	(*Reposition Request#3*)
	(*Pick Up repo*)
	IF (MAIN.R4.Peripheral_Req.2 AND (MAIN.R4.Task_ID_Ack=Pickup_Fix102))
		THEN
			Repo_Reqs.2:= TRUE;
	END_IF;

	(*Reposition Request#4*)
	IF FALSE
		THEN
			Repo_Reqs.3:= TRUE;
	END_IF;

	(*Reposition Request#5*)
	IF FALSE
		THEN
			Repo_Reqs.4:= TRUE;
	END_IF;

	(*Reposition Request#6*)
	IF FALSE
		THEN
			Repo_Reqs.5:= TRUE;
	END_IF;

	(*Reposition Request#7*)
	IF FALSE
		THEN
			Repo_Reqs.6:= TRUE;
	END_IF;

	(*Reposition Request#8*)
	IF FALSE
		THEN
			Repo_Reqs.7:= TRUE;
	END_IF;

	(*Reset All Reposition Acks At the End Of Cycle*)
	IF Cycle_Complete
		THEN
			Repo_Reqs:= 0;
	END_IF;

(*------------------------- Reposition Acks ---------------------*)
	Repo_Ack.0:= Repo_Reqs.0 AND Tool_At_Load.0;   (*Drop Off*)
	Repo_Ack.1:= Repo_Reqs.1 AND FALSE;            (*Inspection*)
	Repo_Ack.2:= Repo_Reqs.2 AND Tool_At_Unload.1; (*Pick Up*)
	Repo_Ack.3:= Repo_Reqs.3 AND FALSE;
	Repo_Ack.4:= Repo_Reqs.4 AND FALSE;
	Repo_Ack.5:= Repo_Reqs.5 AND FALSE;
	Repo_Ack.6:= Repo_Reqs.6 AND FALSE;
	Repo_Ack.7:= Repo_Reqs.7 AND FALSE;
END_ACTION

ACTION ValveBank1:


(*+++++++++++THIS AREA IS CUSTOM PER INSTALLATION AND WILL HAVE TO BE MODIFIED PER +++++++++++++*)
(*+++++++++++THIS AREA IS CUSTOM PER INSTALLATION AND WILL HAVE TO BE MODIFIED PER +++++++++++++*)
(*+++++++++++THIS AREA IS CUSTOM PER INSTALLATION AND WILL HAVE TO BE MODIFIED PER +++++++++++++*)

(*+++++++++++VALVE BANK 1 +++++++++++++*)
(*+++++++++++VALVE BANK 1 +++++++++++++*)
(*+++++++++++VALVE BANK 1 +++++++++++++*)


	(*Valve 1, A+B*)
	// NOW Pin 1,2 Piped and Labled From Supplier (*TLK*)
		Valve1FB
			(
			Enable_Motion:= Enable_Motion ,
			Enable_Latch:= TRUE,					(*Enabling Runs Valve as detent type (maintained solenoids*)
			Enable_SideA_PreCharge:= FALSE,		(*Enabling Turns Side A PreCharge Active, reset when Side B is energized in Auto*)
			Enable_SideB_PreCharge:= FALSE,		(*Enabling Turns Side B PreCharge Active, reset when Side A is energized in Auto*)
			PreCharge_Time:= T#0.1S,
			Enable_Auto_Commands:= In_Auto,
			Enable_Manual_Commands:= In_Manual AND All_Robots_Clear,
			In_Manual_SideA_Command:= Discrete_In.ManReqs.0,
			In_Manual_SideB_Command:= (Discrete_In.ManReqs.1 OR Discrete_In.Go_Home),
			SideA_Indicator:= (Pin1ADVD AND Pin2ADVD) OR Manual_Ind_HomePrompt,
			SideB_Indicator:= (Pin1RETD AND Pin2RETD),
			TurnOn_SideA_SOL=> N100.Q.0,
			TurnOn_SideB_SOL=> N100.Q.1,
			TurnOn_SideA_Indicator=> Manual_Indicators1.0,
			TurnOn_SideB_Indicator=> Manual_Indicators1.1
			 );
		Valve1FB.In_Auto_SideA_Command:= (*Clamp_Step.1 AND NOT Unclamp_Step.1;*) Clamp_Step.0 AND NOT Unclamp_Step.0;
		Valve1FB.In_Auto_SideB_Command:= (*NOT Clamp_Step.1 AND Unclamp_Step.1;*) NOT Clamp_Step.0 AND Unclamp_Step.0;


	(*Valve 2, A+B*)
	// NOW Clamp 1,2,3,4 Piped and Labled From Supplier (*TLK*)
		Valve2FB
			(
			Enable_Motion:= Enable_Motion ,
			Enable_Latch:= TRUE,					(*Enabling Runs Valve as detent type (maintained solenoids*)
			Enable_SideA_PreCharge:= FALSE,		(*Enabling Turns Side A PreCharge Active, reset when Side B is energized in Auto*)
			Enable_SideB_PreCharge:= FALSE,		(*Enabling Turns Side B PreCharge Active, reset when Side A is energized in Auto*)
			PreCharge_Time:= T#0.10S,
			Enable_Auto_Commands:= In_Auto,
			Enable_Manual_Commands:= In_Manual AND All_Robots_Clear,
			In_Manual_SideA_Command:= (Discrete_In.ManReqs.2 OR Discrete_In.Go_Home),
			In_Manual_SideB_Command:= Discrete_In.ManReqs.3,		
			SideA_Indicator:= (Clamp1ADVD AND Clamp2ADVD AND Clamp3ADVD AND Clamp4ADVD),
			SideB_Indicator:= (Clamp1RETD AND Clamp2RETD AND Clamp3RETD AND Clamp4RETD) OR Manual_Ind_HomePrompt,
			TurnOn_SideA_SOL=> N100.Q.2,
			TurnOn_SideB_SOL=> N100.Q.3,
			TurnOn_SideA_Indicator=> Manual_Indicators1.2,
			TurnOn_SideB_Indicator=> Manual_Indicators1.3
			 );
		Valve2FB.In_Auto_SideA_Command:= (*Clamp_Step.0 AND NOT Unclamp_Step.0;*) Clamp_Step.1 AND NOT Unclamp_Step.1;
		Valve2FB.In_Auto_SideB_Command:= (*NOT Clamp_Step.0 AND Unclamp_Step.0;*) NOT Clamp_Step.1 AND Unclamp_Step.1;


		
		
		
		
		
		
		
		
		
		
		
		
		
		
		
		
		
		
		
	(*Valve 3, A+B*)
	(*spare*)
		Valve3FB
			(
			Enable_Motion:= Enable_Motion ,
			Enable_Latch:= TRUE,					(*Enabling Runs Valve as detent type (maintained solenoids*)
			Enable_SideA_PreCharge:= FALSE,		(*Enabling Turns Side A PreCharge Active, reset when Side B is energized in Auto*)
			Enable_SideB_PreCharge:= FALSE,		(*Enabling Turns Side B PreCharge Active, reset when Side A is energized in Auto*)
			PreCharge_Time:= T#0.10S,
			Enable_Auto_Commands:= In_Auto,
			Enable_Manual_Commands:= In_Manual AND All_Robots_Clear,
			In_Manual_SideA_Command:= Discrete_In.ManReqs.4,
			In_Manual_SideB_Command:= Discrete_In.ManReqs.5,
			SideA_Indicator:= FALSE,
			SideB_Indicator:= FALSE,
			TurnOn_SideA_SOL=> N100.Q.4,
			TurnOn_SideB_SOL=> N100.Q.5,
			TurnOn_SideA_Indicator=> Manual_Indicators1.4,
			TurnOn_SideB_Indicator=> Manual_Indicators1.5
			 );
		Valve3FB.In_Auto_SideA_Command:= FALSE;
		Valve3FB.In_Auto_SideB_Command:= FALSE;



(*end*)
END_ACTION

ACTION ValveBank2:


(*+++++++++++THIS AREA IS CUSTOM PER INSTALLATION AND WILL HAVE TO BE MODIFIED PER +++++++++++++*)
(*+++++++++++THIS AREA IS CUSTOM PER INSTALLATION AND WILL HAVE TO BE MODIFIED PER +++++++++++++*)
(*+++++++++++THIS AREA IS CUSTOM PER INSTALLATION AND WILL HAVE TO BE MODIFIED PER +++++++++++++*)

(*+++++++++++VALVE BANK 2 +++++++++++++*)
(*+++++++++++VALVE BANK 2 +++++++++++++*)
(*+++++++++++VALVE BANK 2 +++++++++++++*)


	(*Valve 17, A+B*)
	(*spare*)
		Valve17FB
			(
			Enable_Motion:= Enable_Motion ,
			Enable_Latch:= TRUE,					(*Enabling Runs Valve as detent type (maintained solenoids*)
			Enable_SideA_PreCharge:= FALSE,		(*Enabling Turns Side A PreCharge Active, reset when Side B is energized in Auto*)
			Enable_SideB_PreCharge:= FALSE,		(*Enabling Turns Side B PreCharge Active, reset when Side A is energized in Auto*)
			PreCharge_Time:= T#0.1S,
			Enable_Auto_Commands:= In_Auto,
			Enable_Manual_Commands:= In_Manual AND All_Robots_Clear,
			In_Manual_SideA_Command:= Discrete_In.ManReqs2.0,
			In_Manual_SideB_Command:= (Discrete_In.ManReqs2.1 OR Discrete_In.Go_Home),
			SideA_Indicator:= FALSE,
			SideB_Indicator:= FALSE,
			TurnOn_SideA_SOL=> N101.Q.0,
			TurnOn_SideB_SOL=> N101.Q.1,
			TurnOn_SideA_Indicator=> Manual_Indicators2.0,
			TurnOn_SideB_Indicator=> Manual_Indicators2.1
			 );
		Valve17FB.In_Auto_SideA_Command:= FALSE;
		Valve17FB.In_Auto_SideB_Command:= FALSE;


	(*Valve 18, A+B*)
	(*spare*)
		Valve18FB
			(
			Enable_Motion:= Enable_Motion ,
			Enable_Latch:= TRUE,					(*Enabling Runs Valve as detent type (maintained solenoids*)
			Enable_SideA_PreCharge:= FALSE,		(*Enabling Turns Side A PreCharge Active, reset when Side B is energized in Auto*)
			Enable_SideB_PreCharge:= FALSE,		(*Enabling Turns Side B PreCharge Active, reset when Side A is energized in Auto*)
			PreCharge_Time:= T#0.10S,
			Enable_Auto_Commands:= In_Auto,
			Enable_Manual_Commands:= In_Manual AND All_Robots_Clear,
			In_Manual_SideA_Command:= Discrete_In.ManReqs2.2,
			In_Manual_SideB_Command:= Discrete_In.ManReqs2.3,
			SideA_Indicator:= FALSE,
			SideB_Indicator:= FALSE,
			TurnOn_SideA_SOL=> N101.Q.2,
			TurnOn_SideB_SOL=> N101.Q.3,
			TurnOn_SideA_Indicator=> Manual_Indicators2.2,
			TurnOn_SideB_Indicator=> Manual_Indicators2.3
			 );
		Valve18FB.In_Auto_SideA_Command:= FALSE;
		Valve18FB.In_Auto_SideB_Command:= FALSE;

	(*Valve 19, A+B*)
	(*spare*)
		Valve19FB
			(
			Enable_Motion:= Enable_Motion ,
			Enable_Latch:= TRUE,					(*Enabling Runs Valve as detent type (maintained solenoids*)
			Enable_SideA_PreCharge:= FALSE,		(*Enabling Turns Side A PreCharge Active, reset when Side B is energized in Auto*)
			Enable_SideB_PreCharge:= FALSE,		(*Enabling Turns Side B PreCharge Active, reset when Side A is energized in Auto*)
			PreCharge_Time:= T#0.10S,
			Enable_Auto_Commands:= In_Auto,
			Enable_Manual_Commands:= In_Manual AND All_Robots_Clear,
			In_Manual_SideA_Command:= Discrete_In.ManReqs2.4,
			In_Manual_SideB_Command:= Discrete_In.ManReqs2.5,
			SideA_Indicator:= FALSE,
			SideB_Indicator:= FALSE,
			TurnOn_SideA_SOL=> N101.Q.4,
			TurnOn_SideB_SOL=> N101.Q.5,
			TurnOn_SideA_Indicator=> Manual_Indicators2.4,
			TurnOn_SideB_Indicator=> Manual_Indicators2.5
			 );
		Valve19FB.In_Auto_SideA_Command:= FALSE;
		Valve19FB.In_Auto_SideB_Command:= FALSE;


	(*Valve 20, A+B*)
	(*spare*)
		Valve20FB
			(
			Enable_Motion:= Enable_Motion ,
			Enable_Latch:= TRUE,					(*Enabling Runs Valve as detent type (maintained solenoids*)
			Enable_SideA_PreCharge:= FALSE,		(*Enabling Turns Side A PreCharge Active, reset when Side B is energized in Auto*)
			Enable_SideB_PreCharge:= FALSE,		(*Enabling Turns Side B PreCharge Active, reset when Side A is energized in Auto*)
			PreCharge_Time:= T#0.10S,
			Enable_Auto_Commands:= In_Auto,
			Enable_Manual_Commands:= In_Manual AND All_Robots_Clear,
			In_Manual_SideA_Command:= Discrete_In.ManReqs2.6,
			In_Manual_SideB_Command:= Discrete_In.ManReqs2.7,
			SideA_Indicator:= FALSE,
			SideB_Indicator:= FALSE,
			TurnOn_SideA_SOL=> N101.Q.6,
			TurnOn_SideB_SOL=> N101.Q.7,
			TurnOn_SideA_Indicator=> Manual_Indicators2.6,
			TurnOn_SideB_Indicator=> Manual_Indicators2.7
			 );
		Valve20FB.In_Auto_SideA_Command:= FALSE;
		Valve20FB.In_Auto_SideB_Command:= FALSE;


	(*Valve 21, A+B*)
	(*spare*)
		Valve21FB
			(
			Enable_Motion:= Enable_Motion ,
			Enable_Latch:= TRUE,					(*Enabling Runs Valve as detent type (maintained solenoids*)
			Enable_SideA_PreCharge:= FALSE,		(*Enabling Turns Side A PreCharge Active, reset when Side B is energized in Auto*)
			Enable_SideB_PreCharge:= FALSE,		(*Enabling Turns Side B PreCharge Active, reset when Side A is energized in Auto*)
			PreCharge_Time:= T#0.10S,
			Enable_Auto_Commands:= In_Auto,
			Enable_Manual_Commands:= In_Manual AND All_Robots_Clear,
			In_Manual_SideA_Command:= Discrete_In.ManReqs2.8,
			In_Manual_SideB_Command:= Discrete_In.ManReqs2.9,
			SideA_Indicator:= FALSE,
			SideB_Indicator:= FALSE,
			TurnOn_SideA_SOL=> N101.Q.8,
			TurnOn_SideB_SOL=> N101.Q.9,
			TurnOn_SideA_Indicator=> Manual_Indicators2.8,
			TurnOn_SideB_Indicator=> Manual_Indicators2.9
			 );
		Valve21FB.In_Auto_SideA_Command:= FALSE;
		Valve21FB.In_Auto_SideB_Command:= FALSE;


	(*Valve 22, A+B*)
	(*spare*)
		Valve22FB
			(
			Enable_Motion:= Enable_Motion ,
			Enable_Latch:= TRUE,					(*Enabling Runs Valve as detent type (maintained solenoids*)
			Enable_SideA_PreCharge:= FALSE,		(*Enabling Turns Side A PreCharge Active, reset when Side B is energized in Auto*)
			Enable_SideB_PreCharge:= FALSE,		(*Enabling Turns Side B PreCharge Active, reset when Side A is energized in Auto*)
			PreCharge_Time:= T#0.10S,
			Enable_Auto_Commands:= In_Auto,
			Enable_Manual_Commands:= In_Manual AND All_Robots_Clear,
			In_Manual_SideA_Command:= Discrete_In.ManReqs2.10,
			In_Manual_SideB_Command:= Discrete_In.ManReqs2.11,
			SideA_Indicator:= FALSE,
			SideB_Indicator:= FALSE,
			TurnOn_SideA_SOL=> N101.Q.10,
			TurnOn_SideB_SOL=> N101.Q.11,
			TurnOn_SideA_Indicator=> Manual_Indicators2.10,
			TurnOn_SideB_Indicator=> Manual_Indicators2.11
			 );
		Valve22FB.In_Auto_SideA_Command:= FALSE;
		Valve22FB.In_Auto_SideB_Command:= FALSE;


	(*Valve 23, A+B*)
	(*spare*)
		Valve23FB
			(
			Enable_Motion:= Enable_Motion ,
			Enable_Latch:= TRUE,					(*Enabling Runs Valve as detent type (maintained solenoids*)
			Enable_SideA_PreCharge:= FALSE,		(*Enabling Turns Side A PreCharge Active, reset when Side B is energized in Auto*)
			Enable_SideB_PreCharge:= FALSE,		(*Enabling Turns Side B PreCharge Active, reset when Side A is energized in Auto*)
			PreCharge_Time:= T#0.10S,
			Enable_Auto_Commands:= In_Auto,
			Enable_Manual_Commands:= In_Manual AND All_Robots_Clear,
			In_Manual_SideA_Command:= Discrete_In.ManReqs2.12,
			In_Manual_SideB_Command:= Discrete_In.ManReqs2.13,
			SideA_Indicator:= FALSE,
			SideB_Indicator:= FALSE,
			TurnOn_SideA_SOL=> N101.Q.12,
			TurnOn_SideB_SOL=> N101.Q.13,
			TurnOn_SideA_Indicator=> Manual_Indicators2.12,
			TurnOn_SideB_Indicator=> Manual_Indicators2.13
			 );
		Valve23FB.In_Auto_SideA_Command:= FALSE;
		Valve23FB.In_Auto_SideB_Command:= FALSE;


	(*Valve 24, A+B*)
	(*spare*)
		Valve24FB
			(
			Enable_Motion:= Enable_Motion ,
			Enable_Latch:= TRUE,					(*Enabling Runs Valve as detent type (maintained solenoids*)
			Enable_SideA_PreCharge:= FALSE,		(*Enabling Turns Side A PreCharge Active, reset when Side B is energized in Auto*)
			Enable_SideB_PreCharge:= FALSE,		(*Enabling Turns Side B PreCharge Active, reset when Side A is energized in Auto*)
			PreCharge_Time:= T#0.10S,
			Enable_Auto_Commands:= In_Auto,
			Enable_Manual_Commands:= In_Manual AND All_Robots_Clear,
			In_Manual_SideA_Command:= Discrete_In.ManReqs2.14,
			In_Manual_SideB_Command:= Discrete_In.ManReqs2.15,
			SideA_Indicator:= FALSE,
			SideB_Indicator:= FALSE,
			TurnOn_SideA_SOL=> N101.Q.14,
			TurnOn_SideB_SOL=> N101.Q.15,
			TurnOn_SideA_Indicator=> Manual_Indicators2.14,
			TurnOn_SideB_Indicator=> Manual_Indicators2.15
			 );
		Valve24FB.In_Auto_SideA_Command:= FALSE;
		Valve24FB.In_Auto_SideB_Command:= FALSE;


	(*Valve 25, A+B*)
	(*spare*)
		Valve25FB
			(
			Enable_Motion:= Enable_Motion ,
			Enable_Latch:= TRUE,					(*Enabling Runs Valve as detent type (maintained solenoids*)
			Enable_SideA_PreCharge:= FALSE,		(*Enabling Turns Side A PreCharge Active, reset when Side B is energized in Auto*)
			Enable_SideB_PreCharge:= FALSE,		(*Enabling Turns Side B PreCharge Active, reset when Side A is energized in Auto*)
			PreCharge_Time:= T#0.10S,
			Enable_Auto_Commands:= In_Auto,
			Enable_Manual_Commands:= In_Manual AND All_Robots_Clear,
			In_Manual_SideA_Command:= Discrete_In.ManReqs2.16,
			In_Manual_SideB_Command:= Discrete_In.ManReqs2.17,
			SideA_Indicator:= FALSE,
			SideB_Indicator:= FALSE,
			TurnOn_SideA_SOL=> N101.Q.16,
			TurnOn_SideB_SOL=> N101.Q.17,
			TurnOn_SideA_Indicator=> Manual_Indicators2.16,
			TurnOn_SideB_Indicator=> Manual_Indicators2.17
			 );
		Valve25FB.In_Auto_SideA_Command:= FALSE;
		Valve25FB.In_Auto_SideB_Command:= FALSE;


	(*Valve 26, A+B*)
	(*spare*)
		Valve26FB
			(
			Enable_Motion:= Enable_Motion ,
			Enable_Latch:= TRUE,					(*Enabling Runs Valve as detent type (maintained solenoids*)
			Enable_SideA_PreCharge:= FALSE,		(*Enabling Turns Side A PreCharge Active, reset when Side B is energized in Auto*)
			Enable_SideB_PreCharge:= FALSE,		(*Enabling Turns Side B PreCharge Active, reset when Side A is energized in Auto*)
			PreCharge_Time:= T#0.10S,
			Enable_Auto_Commands:= In_Auto,
			Enable_Manual_Commands:= In_Manual AND All_Robots_Clear,
			In_Manual_SideA_Command:= Discrete_In.ManReqs2.18,
			In_Manual_SideB_Command:= Discrete_In.ManReqs2.19,
			SideA_Indicator:= FALSE,
			SideB_Indicator:= FALSE,
			TurnOn_SideA_SOL=> N101.Q.18,
			TurnOn_SideB_SOL=> N101.Q.19,
			TurnOn_SideA_Indicator=> Manual_Indicators2.18,
			TurnOn_SideB_Indicator=> Manual_Indicators2.19
			 );
		Valve26FB.In_Auto_SideA_Command:= FALSE;
		Valve26FB.In_Auto_SideB_Command:= FALSE;


	(*Valve 27, A+B*)
	(*spare*)
		Valve27FB
			(
			Enable_Motion:= Enable_Motion ,
			Enable_Latch:= TRUE,					(*Enabling Runs Valve as detent type (maintained solenoids*)
			Enable_SideA_PreCharge:= FALSE,		(*Enabling Turns Side A PreCharge Active, reset when Side B is energized in Auto*)
			Enable_SideB_PreCharge:= FALSE,		(*Enabling Turns Side B PreCharge Active, reset when Side A is energized in Auto*)
			PreCharge_Time:= T#0.10S,
			Enable_Auto_Commands:= In_Auto,
			Enable_Manual_Commands:= In_Manual AND All_Robots_Clear,
			In_Manual_SideA_Command:= Discrete_In.ManReqs2.20,
			In_Manual_SideB_Command:= Discrete_In.ManReqs2.21,
			SideA_Indicator:= FALSE,
			SideB_Indicator:= FALSE,
			TurnOn_SideA_SOL=> N101.Q.20,
			TurnOn_SideB_SOL=> N101.Q.21,
			TurnOn_SideA_Indicator=> Manual_Indicators2.20,
			TurnOn_SideB_Indicator=> Manual_Indicators2.21
			 );
		Valve27FB.In_Auto_SideA_Command:= FALSE;
		Valve27FB.In_Auto_SideB_Command:= FALSE;


	(*Valve 28, A+B*)
	(*spare*)
		Valve28FB
			(
			Enable_Motion:= Enable_Motion ,
			Enable_Latch:= TRUE,					(*Enabling Runs Valve as detent type (maintained solenoids*)
			Enable_SideA_PreCharge:= FALSE,		(*Enabling Turns Side A PreCharge Active, reset when Side B is energized in Auto*)
			Enable_SideB_PreCharge:= FALSE,		(*Enabling Turns Side B PreCharge Active, reset when Side A is energized in Auto*)
			PreCharge_Time:= T#0.10S,
			Enable_Auto_Commands:= In_Auto,
			Enable_Manual_Commands:= In_Manual AND All_Robots_Clear,
			In_Manual_SideA_Command:= Discrete_In.ManReqs2.22,
			In_Manual_SideB_Command:= Discrete_In.ManReqs2.23,
			SideA_Indicator:= FALSE,
			SideB_Indicator:= FALSE,
			TurnOn_SideA_SOL=> N101.Q.22,
			TurnOn_SideB_SOL=> N101.Q.23,
			TurnOn_SideA_Indicator=> Manual_Indicators2.22,
			TurnOn_SideB_Indicator=> Manual_Indicators2.23
			 );
		Valve28FB.In_Auto_SideA_Command:= FALSE;
		Valve28FB.In_Auto_SideB_Command:= FALSE;


	(*Valve 29, A+B*)
	(*spare*)
		Valve29FB
			(
			Enable_Motion:= Enable_Motion ,
			Enable_Latch:= TRUE,					(*Enabling Runs Valve as detent type (maintained solenoids*)
			Enable_SideA_PreCharge:= FALSE,		(*Enabling Turns Side A PreCharge Active, reset when Side B is energized in Auto*)
			Enable_SideB_PreCharge:= FALSE,		(*Enabling Turns Side B PreCharge Active, reset when Side A is energized in Auto*)
			PreCharge_Time:= T#0.10S,
			Enable_Auto_Commands:= In_Auto,
			Enable_Manual_Commands:= In_Manual AND All_Robots_Clear,
			In_Manual_SideA_Command:= Discrete_In.ManReqs2.24,
			In_Manual_SideB_Command:= Discrete_In.ManReqs2.25,
			SideA_Indicator:= FALSE,
			SideB_Indicator:= FALSE,
			TurnOn_SideA_SOL=> N101.Q.24,
			TurnOn_SideB_SOL=> N101.Q.25,
			TurnOn_SideA_Indicator=> Manual_Indicators2.24,
			TurnOn_SideB_Indicator=> Manual_Indicators2.25
			 );
		Valve29FB.In_Auto_SideA_Command:= FALSE;
		Valve29FB.In_Auto_SideB_Command:= FALSE;


	(*Valve 30, A+B*)
	(*spare*)
		Valve30FB
			(
			Enable_Motion:= Enable_Motion ,
			Enable_Latch:= TRUE,					(*Enabling Runs Valve as detent type (maintained solenoids*)
			Enable_SideA_PreCharge:= FALSE,		(*Enabling Turns Side A PreCharge Active, reset when Side B is energized in Auto*)
			Enable_SideB_PreCharge:= FALSE,		(*Enabling Turns Side B PreCharge Active, reset when Side A is energized in Auto*)
			PreCharge_Time:= T#0.10S,
			Enable_Auto_Commands:= In_Auto,
			Enable_Manual_Commands:= In_Manual AND All_Robots_Clear,
			In_Manual_SideA_Command:= Discrete_In.ManReqs2.26,
			In_Manual_SideB_Command:= Discrete_In.ManReqs2.27,
			SideA_Indicator:= FALSE,
			SideB_Indicator:= FALSE,
			TurnOn_SideA_SOL=> N101.Q.26,
			TurnOn_SideB_SOL=> N101.Q.27,
			TurnOn_SideA_Indicator=> Manual_Indicators2.26,
			TurnOn_SideB_Indicator=> Manual_Indicators2.27
			 );
		Valve30FB.In_Auto_SideA_Command:= FALSE;
		Valve30FB.In_Auto_SideB_Command:= FALSE;


	(*Valve 31, A+B*)
	(*spare*)
		Valve31FB
			(
			Enable_Motion:= Enable_Motion ,
			Enable_Latch:= TRUE,					(*Enabling Runs Valve as detent type (maintained solenoids*)
			Enable_SideA_PreCharge:= FALSE,		(*Enabling Turns Side A PreCharge Active, reset when Side B is energized in Auto*)
			Enable_SideB_PreCharge:= FALSE,		(*Enabling Turns Side B PreCharge Active, reset when Side A is energized in Auto*)
			PreCharge_Time:= T#0.10S,
			Enable_Auto_Commands:= In_Auto,
			Enable_Manual_Commands:= In_Manual AND All_Robots_Clear,
			In_Manual_SideA_Command:= Discrete_In.ManReqs2.28,
			In_Manual_SideB_Command:= Discrete_In.ManReqs2.29,
			SideA_Indicator:= FALSE,
			SideB_Indicator:= FALSE,
			TurnOn_SideA_SOL=> N101.Q.28,
			TurnOn_SideB_SOL=> N101.Q.29,
			TurnOn_SideA_Indicator=> Manual_Indicators2.28,
			TurnOn_SideB_Indicator=> Manual_Indicators2.29
			 );
		Valve31FB.In_Auto_SideA_Command:= FALSE;
		Valve31FB.In_Auto_SideB_Command:= FALSE;


	(*Valve 32, A+B*)
	(*spare*)
		Valve32FB
			(
			Enable_Motion:= Enable_Motion ,
			Enable_Latch:= TRUE,					(*Enabling Runs Valve as detent type (maintained solenoids*)
			Enable_SideA_PreCharge:= FALSE,		(*Enabling Turns Side A PreCharge Active, reset when Side B is energized in Auto*)
			Enable_SideB_PreCharge:= FALSE,		(*Enabling Turns Side B PreCharge Active, reset when Side A is energized in Auto*)
			PreCharge_Time:= T#0.10S,
			Enable_Auto_Commands:= In_Auto,
			Enable_Manual_Commands:= In_Manual AND All_Robots_Clear,
			In_Manual_SideA_Command:= Discrete_In.ManReqs2.30,
			In_Manual_SideB_Command:= Discrete_In.ManReqs2.31,
			SideA_Indicator:= FALSE,
			SideB_Indicator:= FALSE,
			TurnOn_SideA_SOL=> N101.Q.30,
			TurnOn_SideB_SOL=> N101.Q.31,
			TurnOn_SideA_Indicator=> Manual_Indicators2.30,
			TurnOn_SideB_Indicator=> Manual_Indicators2.31
			 );
		Valve32FB.In_Auto_SideA_Command:= FALSE;
		Valve32FB.In_Auto_SideB_Command:= FALSE;




















(*end*)
END_ACTION

ACTION ValveBank3:


(*+++++++++++THIS AREA IS CUSTOM PER INSTALLATION AND WILL HAVE TO BE MODIFIED PER +++++++++++++*)
(*+++++++++++THIS AREA IS CUSTOM PER INSTALLATION AND WILL HAVE TO BE MODIFIED PER +++++++++++++*)
(*+++++++++++THIS AREA IS CUSTOM PER INSTALLATION AND WILL HAVE TO BE MODIFIED PER +++++++++++++*)

(*+++++++++++VALVE BANK 3 +++++++++++++*)
(*+++++++++++VALVE BANK 3 +++++++++++++*)
(*+++++++++++VALVE BANK 3 +++++++++++++*)


	(*Valve 33, A+B*)
	(*spare*)
		Valve33FB
			(
			Enable_Motion:= Enable_Motion ,
			Enable_Latch:= TRUE,					(*Enabling Runs Valve as detent type (maintained solenoids*)
			Enable_SideA_PreCharge:= FALSE,		(*Enabling Turns Side A PreCharge Active, reset when Side B is energized in Auto*)
			Enable_SideB_PreCharge:= FALSE,		(*Enabling Turns Side B PreCharge Active, reset when Side A is energized in Auto*)
			PreCharge_Time:= T#0.1S,
			Enable_Auto_Commands:= In_Auto,
			Enable_Manual_Commands:= In_Manual AND All_Robots_Clear,
			In_Manual_SideA_Command:= Discrete_In.ManReqs3.0,
			In_Manual_SideB_Command:= (Discrete_In.ManReqs3.1 OR Discrete_In.Go_Home),
			SideA_Indicator:= FALSE,
			SideB_Indicator:= FALSE,
			TurnOn_SideA_SOL=> N102.Q.0,
			TurnOn_SideB_SOL=> N102.Q.1,
			TurnOn_SideA_Indicator=> Manual_Indicators3.0,
			TurnOn_SideB_Indicator=> Manual_Indicators3.1
			 );
		Valve33FB.In_Auto_SideA_Command:= FALSE;
		Valve33FB.In_Auto_SideB_Command:= FALSE;


	(*Valve 34, A+B*)
	(*spare*)
		Valve34FB
			(
			Enable_Motion:= Enable_Motion ,
			Enable_Latch:= TRUE,					(*Enabling Runs Valve as detent type (maintained solenoids*)
			Enable_SideA_PreCharge:= FALSE,		(*Enabling Turns Side A PreCharge Active, reset when Side B is energized in Auto*)
			Enable_SideB_PreCharge:= FALSE,		(*Enabling Turns Side B PreCharge Active, reset when Side A is energized in Auto*)
			PreCharge_Time:= T#0.10S,
			Enable_Auto_Commands:= In_Auto,
			Enable_Manual_Commands:= In_Manual AND All_Robots_Clear,
			In_Manual_SideA_Command:= Discrete_In.ManReqs3.2,
			In_Manual_SideB_Command:= Discrete_In.ManReqs3.3,
			SideA_Indicator:= FALSE,
			SideB_Indicator:= FALSE,
			TurnOn_SideA_SOL=> N102.Q.2,
			TurnOn_SideB_SOL=> N102.Q.3,
			TurnOn_SideA_Indicator=> Manual_Indicators3.2,
			TurnOn_SideB_Indicator=> Manual_Indicators3.3
			 );
		Valve34FB.In_Auto_SideA_Command:= FALSE;
		Valve34FB.In_Auto_SideB_Command:= FALSE;


	(*Valve 35, A+B*)
	(*spare*)
		Valve35FB
			(
			Enable_Motion:= Enable_Motion ,
			Enable_Latch:= TRUE,					(*Enabling Runs Valve as detent type (maintained solenoids*)
			Enable_SideA_PreCharge:= FALSE,		(*Enabling Turns Side A PreCharge Active, reset when Side B is energized in Auto*)
			Enable_SideB_PreCharge:= FALSE,		(*Enabling Turns Side B PreCharge Active, reset when Side A is energized in Auto*)
			PreCharge_Time:= T#0.10S,
			Enable_Auto_Commands:= In_Auto,
			Enable_Manual_Commands:= In_Manual AND All_Robots_Clear,
			In_Manual_SideA_Command:= Discrete_In.ManReqs3.4,
			In_Manual_SideB_Command:= Discrete_In.ManReqs3.5,
			SideA_Indicator:= FALSE,
			SideB_Indicator:= FALSE,
			TurnOn_SideA_SOL=> N102.Q.4,
			TurnOn_SideB_SOL=> N102.Q.5,
			TurnOn_SideA_Indicator=> Manual_Indicators3.4,
			TurnOn_SideB_Indicator=> Manual_Indicators3.5
			 );
		Valve35FB.In_Auto_SideA_Command:= FALSE;
		Valve35FB.In_Auto_SideB_Command:= FALSE;


	(*Valve 36, A+B*)
	(*spare*)
		Valve36FB
			(
			Enable_Motion:= Enable_Motion ,
			Enable_Latch:= TRUE,					(*Enabling Runs Valve as detent type (maintained solenoids*)
			Enable_SideA_PreCharge:= FALSE,		(*Enabling Turns Side A PreCharge Active, reset when Side B is energized in Auto*)
			Enable_SideB_PreCharge:= FALSE,		(*Enabling Turns Side B PreCharge Active, reset when Side A is energized in Auto*)
			PreCharge_Time:= T#0.10S,
			Enable_Auto_Commands:= In_Auto,
			Enable_Manual_Commands:= In_Manual AND All_Robots_Clear,
			In_Manual_SideA_Command:= Discrete_In.ManReqs3.6,
			In_Manual_SideB_Command:= Discrete_In.ManReqs3.7,
			SideA_Indicator:= FALSE,
			SideB_Indicator:= FALSE,
			TurnOn_SideA_SOL=> N102.Q.6,
			TurnOn_SideB_SOL=> N102.Q.7,
			TurnOn_SideA_Indicator=> Manual_Indicators3.6,
			TurnOn_SideB_Indicator=> Manual_Indicators3.7
			 );
		Valve36FB.In_Auto_SideA_Command:= FALSE;
		Valve36FB.In_Auto_SideB_Command:= FALSE;


	(*Valve 37, A+B*)
	(*spare*)
		Valve37FB
			(
			Enable_Motion:= Enable_Motion ,
			Enable_Latch:= TRUE,					(*Enabling Runs Valve as detent type (maintained solenoids*)
			Enable_SideA_PreCharge:= FALSE,		(*Enabling Turns Side A PreCharge Active, reset when Side B is energized in Auto*)
			Enable_SideB_PreCharge:= FALSE,		(*Enabling Turns Side B PreCharge Active, reset when Side A is energized in Auto*)
			PreCharge_Time:= T#0.10S,
			Enable_Auto_Commands:= In_Auto,
			Enable_Manual_Commands:= In_Manual AND All_Robots_Clear,
			In_Manual_SideA_Command:= Discrete_In.ManReqs3.8,
			In_Manual_SideB_Command:= Discrete_In.ManReqs3.9,
			SideA_Indicator:= FALSE,
			SideB_Indicator:= FALSE,
			TurnOn_SideA_SOL=> N102.Q.8,
			TurnOn_SideB_SOL=> N102.Q.9,
			TurnOn_SideA_Indicator=> Manual_Indicators3.8,
			TurnOn_SideB_Indicator=> Manual_Indicators3.9
			 );
		Valve37FB.In_Auto_SideA_Command:= FALSE;
		Valve37FB.In_Auto_SideB_Command:= FALSE;


	(*Valve 38, A+B*)
	(*spare*)
		Valve38FB
			(
			Enable_Motion:= Enable_Motion ,
			Enable_Latch:= TRUE,					(*Enabling Runs Valve as detent type (maintained solenoids*)
			Enable_SideA_PreCharge:= FALSE,		(*Enabling Turns Side A PreCharge Active, reset when Side B is energized in Auto*)
			Enable_SideB_PreCharge:= FALSE,		(*Enabling Turns Side B PreCharge Active, reset when Side A is energized in Auto*)
			PreCharge_Time:= T#0.10S,
			Enable_Auto_Commands:= In_Auto,
			Enable_Manual_Commands:= In_Manual AND All_Robots_Clear,
			In_Manual_SideA_Command:= Discrete_In.ManReqs3.10,
			In_Manual_SideB_Command:= Discrete_In.ManReqs3.11,
			SideA_Indicator:= FALSE,
			SideB_Indicator:= FALSE,
			TurnOn_SideA_SOL=> N102.Q.10,
			TurnOn_SideB_SOL=> N102.Q.11,
			TurnOn_SideA_Indicator=> Manual_Indicators3.10,
			TurnOn_SideB_Indicator=> Manual_Indicators3.11
			 );
		Valve38FB.In_Auto_SideA_Command:= FALSE;
		Valve38FB.In_Auto_SideB_Command:= FALSE;


	(*Valve 39, A+B*)
	(*spare*)
		Valve39FB
			(
			Enable_Motion:= Enable_Motion ,
			Enable_Latch:= TRUE,					(*Enabling Runs Valve as detent type (maintained solenoids*)
			Enable_SideA_PreCharge:= FALSE,		(*Enabling Turns Side A PreCharge Active, reset when Side B is energized in Auto*)
			Enable_SideB_PreCharge:= FALSE,		(*Enabling Turns Side B PreCharge Active, reset when Side A is energized in Auto*)
			PreCharge_Time:= T#0.10S,
			Enable_Auto_Commands:= In_Auto,
			Enable_Manual_Commands:= In_Manual AND All_Robots_Clear,
			In_Manual_SideA_Command:= Discrete_In.ManReqs3.12,
			In_Manual_SideB_Command:= Discrete_In.ManReqs3.13,
			SideA_Indicator:= FALSE,
			SideB_Indicator:= FALSE,
			TurnOn_SideA_SOL=> N102.Q.12,
			TurnOn_SideB_SOL=> N102.Q.13,
			TurnOn_SideA_Indicator=> Manual_Indicators3.12,
			TurnOn_SideB_Indicator=> Manual_Indicators3.13
			 );
		Valve39FB.In_Auto_SideA_Command:= FALSE;
		Valve39FB.In_Auto_SideB_Command:= FALSE;


	(*Valve 40, A+B*)
	(*spare*)
		Valve40FB
			(
			Enable_Motion:= Enable_Motion ,
			Enable_Latch:= TRUE,					(*Enabling Runs Valve as detent type (maintained solenoids*)
			Enable_SideA_PreCharge:= FALSE,		(*Enabling Turns Side A PreCharge Active, reset when Side B is energized in Auto*)
			Enable_SideB_PreCharge:= FALSE,		(*Enabling Turns Side B PreCharge Active, reset when Side A is energized in Auto*)
			PreCharge_Time:= T#0.10S,
			Enable_Auto_Commands:= In_Auto,
			Enable_Manual_Commands:= In_Manual AND All_Robots_Clear,
			In_Manual_SideA_Command:= Discrete_In.ManReqs3.14,
			In_Manual_SideB_Command:= Discrete_In.ManReqs3.15,
			SideA_Indicator:= FALSE,
			SideB_Indicator:= FALSE,
			TurnOn_SideA_SOL=> N102.Q.14,
			TurnOn_SideB_SOL=> N102.Q.15,
			TurnOn_SideA_Indicator=> Manual_Indicators3.14,
			TurnOn_SideB_Indicator=> Manual_Indicators3.15
			 );
		Valve40FB.In_Auto_SideA_Command:= FALSE;
		Valve40FB.In_Auto_SideB_Command:= FALSE;


	(*Valve 41, A+B*)
	(*spare*)
		Valve41FB
			(
			Enable_Motion:= Enable_Motion ,
			Enable_Latch:= TRUE,					(*Enabling Runs Valve as detent type (maintained solenoids*)
			Enable_SideA_PreCharge:= FALSE,		(*Enabling Turns Side A PreCharge Active, reset when Side B is energized in Auto*)
			Enable_SideB_PreCharge:= FALSE,		(*Enabling Turns Side B PreCharge Active, reset when Side A is energized in Auto*)
			PreCharge_Time:= T#0.10S,
			Enable_Auto_Commands:= In_Auto,
			Enable_Manual_Commands:= In_Manual AND All_Robots_Clear,
			In_Manual_SideA_Command:= Discrete_In.ManReqs3.16,
			In_Manual_SideB_Command:= Discrete_In.ManReqs3.17,
			SideA_Indicator:= FALSE,
			SideB_Indicator:= FALSE,
			TurnOn_SideA_SOL=> N102.Q.16,
			TurnOn_SideB_SOL=> N102.Q.17,
			TurnOn_SideA_Indicator=> Manual_Indicators3.16,
			TurnOn_SideB_Indicator=> Manual_Indicators3.17
			 );
		Valve41FB.In_Auto_SideA_Command:= FALSE;
		Valve41FB.In_Auto_SideB_Command:= FALSE;


	(*Valve 42, A+B*)
	(*spare*)
		Valve42FB
			(
			Enable_Motion:= Enable_Motion ,
			Enable_Latch:= TRUE,					(*Enabling Runs Valve as detent type (maintained solenoids*)
			Enable_SideA_PreCharge:= FALSE,		(*Enabling Turns Side A PreCharge Active, reset when Side B is energized in Auto*)
			Enable_SideB_PreCharge:= FALSE,		(*Enabling Turns Side B PreCharge Active, reset when Side A is energized in Auto*)
			PreCharge_Time:= T#0.10S,
			Enable_Auto_Commands:= In_Auto,
			Enable_Manual_Commands:= In_Manual AND All_Robots_Clear,
			In_Manual_SideA_Command:= Discrete_In.ManReqs3.18,
			In_Manual_SideB_Command:= Discrete_In.ManReqs3.19,
			SideA_Indicator:= FALSE,
			SideB_Indicator:= FALSE,
			TurnOn_SideA_SOL=> N102.Q.18,
			TurnOn_SideB_SOL=> N102.Q.19,
			TurnOn_SideA_Indicator=> Manual_Indicators3.18,
			TurnOn_SideB_Indicator=> Manual_Indicators3.19
			 );
		Valve42FB.In_Auto_SideA_Command:= FALSE;
		Valve42FB.In_Auto_SideB_Command:= FALSE;


	(*Valve 43, A+B*)
	(*spare*)
		Valve43FB
			(
			Enable_Motion:= Enable_Motion ,
			Enable_Latch:= TRUE,					(*Enabling Runs Valve as detent type (maintained solenoids*)
			Enable_SideA_PreCharge:= FALSE,		(*Enabling Turns Side A PreCharge Active, reset when Side B is energized in Auto*)
			Enable_SideB_PreCharge:= FALSE,		(*Enabling Turns Side B PreCharge Active, reset when Side A is energized in Auto*)
			PreCharge_Time:= T#0.10S,
			Enable_Auto_Commands:= In_Auto,
			Enable_Manual_Commands:= In_Manual AND All_Robots_Clear,
			In_Manual_SideA_Command:= Discrete_In.ManReqs3.20,
			In_Manual_SideB_Command:= Discrete_In.ManReqs3.21,
			SideA_Indicator:= FALSE,
			SideB_Indicator:= FALSE,
			TurnOn_SideA_SOL=> N102.Q.20,
			TurnOn_SideB_SOL=> N102.Q.21,
			TurnOn_SideA_Indicator=> Manual_Indicators3.20,
			TurnOn_SideB_Indicator=> Manual_Indicators3.21
			 );
		Valve43FB.In_Auto_SideA_Command:= FALSE;
		Valve43FB.In_Auto_SideB_Command:= FALSE;


	(*Valve 44, A+B*)
	(*spare*)
		Valve44FB
			(
			Enable_Motion:= Enable_Motion ,
			Enable_Latch:= TRUE,					(*Enabling Runs Valve as detent type (maintained solenoids*)
			Enable_SideA_PreCharge:= FALSE,		(*Enabling Turns Side A PreCharge Active, reset when Side B is energized in Auto*)
			Enable_SideB_PreCharge:= FALSE,		(*Enabling Turns Side B PreCharge Active, reset when Side A is energized in Auto*)
			PreCharge_Time:= T#0.10S,
			Enable_Auto_Commands:= In_Auto,
			Enable_Manual_Commands:= In_Manual AND All_Robots_Clear,
			In_Manual_SideA_Command:= Discrete_In.ManReqs3.22,
			In_Manual_SideB_Command:= Discrete_In.ManReqs3.23,
			SideA_Indicator:= FALSE,
			SideB_Indicator:= FALSE,
			TurnOn_SideA_SOL=> N102.Q.22,
			TurnOn_SideB_SOL=> N102.Q.23,
			TurnOn_SideA_Indicator=> Manual_Indicators3.22,
			TurnOn_SideB_Indicator=> Manual_Indicators3.23
			 );
		Valve44FB.In_Auto_SideA_Command:= FALSE;
		Valve44FB.In_Auto_SideB_Command:= FALSE;


	(*Valve 45, A+B*)
	(*spare*)
		Valve45FB
			(
			Enable_Motion:= Enable_Motion ,
			Enable_Latch:= TRUE,					(*Enabling Runs Valve as detent type (maintained solenoids*)
			Enable_SideA_PreCharge:= FALSE,		(*Enabling Turns Side A PreCharge Active, reset when Side B is energized in Auto*)
			Enable_SideB_PreCharge:= FALSE,		(*Enabling Turns Side B PreCharge Active, reset when Side A is energized in Auto*)
			PreCharge_Time:= T#0.10S,
			Enable_Auto_Commands:= In_Auto,
			Enable_Manual_Commands:= In_Manual AND All_Robots_Clear,
			In_Manual_SideA_Command:= Discrete_In.ManReqs3.24,
			In_Manual_SideB_Command:= Discrete_In.ManReqs3.25,
			SideA_Indicator:= FALSE,
			SideB_Indicator:= FALSE,
			TurnOn_SideA_SOL=> N102.Q.24,
			TurnOn_SideB_SOL=> N102.Q.25,
			TurnOn_SideA_Indicator=> Manual_Indicators3.24,
			TurnOn_SideB_Indicator=> Manual_Indicators3.25
			 );
		Valve45FB.In_Auto_SideA_Command:= FALSE;
		Valve45FB.In_Auto_SideB_Command:= FALSE;


	(*Valve 46, A+B*)
	(*spare*)
		Valve46FB
			(
			Enable_Motion:= Enable_Motion ,
			Enable_Latch:= TRUE,					(*Enabling Runs Valve as detent type (maintained solenoids*)
			Enable_SideA_PreCharge:= FALSE,		(*Enabling Turns Side A PreCharge Active, reset when Side B is energized in Auto*)
			Enable_SideB_PreCharge:= FALSE,		(*Enabling Turns Side B PreCharge Active, reset when Side A is energized in Auto*)
			PreCharge_Time:= T#0.10S,
			Enable_Auto_Commands:= In_Auto,
			Enable_Manual_Commands:= In_Manual AND All_Robots_Clear,
			In_Manual_SideA_Command:= Discrete_In.ManReqs3.26,
			In_Manual_SideB_Command:= Discrete_In.ManReqs3.27,
			SideA_Indicator:= FALSE,
			SideB_Indicator:= FALSE,
			TurnOn_SideA_SOL=> N102.Q.26,
			TurnOn_SideB_SOL=> N102.Q.27,
			TurnOn_SideA_Indicator=> Manual_Indicators3.26,
			TurnOn_SideB_Indicator=> Manual_Indicators3.27
			 );
		Valve46FB.In_Auto_SideA_Command:= FALSE;
		Valve46FB.In_Auto_SideB_Command:= FALSE;


	(*Valve 47, A+B*)
	(*spare*)
		Valve47FB
			(
			Enable_Motion:= Enable_Motion ,
			Enable_Latch:= TRUE,					(*Enabling Runs Valve as detent type (maintained solenoids*)
			Enable_SideA_PreCharge:= FALSE,		(*Enabling Turns Side A PreCharge Active, reset when Side B is energized in Auto*)
			Enable_SideB_PreCharge:= FALSE,		(*Enabling Turns Side B PreCharge Active, reset when Side A is energized in Auto*)
			PreCharge_Time:= T#0.10S,
			Enable_Auto_Commands:= In_Auto,
			Enable_Manual_Commands:= In_Manual AND All_Robots_Clear,
			In_Manual_SideA_Command:= Discrete_In.ManReqs3.28,
			In_Manual_SideB_Command:= Discrete_In.ManReqs3.29,
			SideA_Indicator:= FALSE,
			SideB_Indicator:= FALSE,
			TurnOn_SideA_SOL=> N102.Q.28,
			TurnOn_SideB_SOL=> N102.Q.29,
			TurnOn_SideA_Indicator=> Manual_Indicators3.28,
			TurnOn_SideB_Indicator=> Manual_Indicators3.29
			 );
		Valve47FB.In_Auto_SideA_Command:= FALSE;
		Valve47FB.In_Auto_SideB_Command:= FALSE;


	(*Valve 48, A+B*)
	(*spare*)
		Valve48FB
			(
			Enable_Motion:= Enable_Motion ,
			Enable_Latch:= TRUE,					(*Enabling Runs Valve as detent type (maintained solenoids*)
			Enable_SideA_PreCharge:= FALSE,		(*Enabling Turns Side A PreCharge Active, reset when Side B is energized in Auto*)
			Enable_SideB_PreCharge:= FALSE,		(*Enabling Turns Side B PreCharge Active, reset when Side A is energized in Auto*)
			PreCharge_Time:= T#0.10S,
			Enable_Auto_Commands:= In_Auto,
			Enable_Manual_Commands:= In_Manual AND All_Robots_Clear,
			In_Manual_SideA_Command:= Discrete_In.ManReqs3.30,
			In_Manual_SideB_Command:= Discrete_In.ManReqs3.31,
			SideA_Indicator:= FALSE,
			SideB_Indicator:= FALSE,
			TurnOn_SideA_SOL=> N102.Q.30,
			TurnOn_SideB_SOL=> N102.Q.31,
			TurnOn_SideA_Indicator=> Manual_Indicators3.30,
			TurnOn_SideB_Indicator=> Manual_Indicators3.31
			 );
		Valve48FB.In_Auto_SideA_Command:= FALSE;
		Valve48FB.In_Auto_SideB_Command:= FALSE;


























(*end*)
END_ACTION

ACTION Xfer_To_UI:
(*Transfer General Status of Fixture and I/O Images for Display On HMI*)
	Discrete_Image.Status:= Status;
	Discrete_Image.CLFaults1:= CLFaults1;
	Discrete_Image.CLFaults2:= CLFaults2;
	Discrete_Image.CLFaults3:= CLFaults3;
	Discrete_Image.CLFaults4:= CLFaults4;
	Discrete_Image.CLFaulted:= CLFaulted;
	Discrete_Image.PPFaults:= PPFaults;
	Discrete_Image.PPFaults1:= PPFaults1;
	Discrete_Image.PPFaults2:= PPFaults2;
	Discrete_Image.PPFaulted:= PPFaulted;
	Discrete_Image.Model_Data:= Model_ID;
	Discrete_Image.ToolID:= Fix_ID;
	Discrete_Image.ProdCount:= Prod_Count_Out;
	Discrete_Image.CycleTime:= Cycle_Time_Out;
	Discrete_Image.PrevCycleTime:= PrevCycle_Time_Out;
	Discrete_Image.LoadTime:= Load_Time_Out;
	Discrete_Image.WeldTime:= Weld_Time_Out;
	Discrete_Image.UnloadTime:= Unload_Time_Out;

	Discrete_Image.InAuto:= In_Auto_Mode;
	Discrete_Image.InManual:= In_Manual_Mode;
	Discrete_Image.ManInds:= Manual_Indicators1;
	Discrete_Image.ManInds2:= Manual_Indicators2;
	Discrete_Image.ManInds3:= Manual_Indicators3;
	Discrete_Image.At_Home:= Tool_At_Home;
	Discrete_Image.Enable_Motion:= Enable_Motion;
	Discrete_Image.All_Sensors_Off:= All_Sensors_Off;
	Discrete_Image.Bypass_ACKS:= Discrete_In.Bypass_REQS;
	Discrete_Image.CustomApplication_ACKS:= Discrete_In.CustomApplication_REQS;
	Discrete_Image.Fixture_Allow_Model_Change:= Fixture_Allow_Model_Change;
	Discrete_Image.NodeLayout:=NodeLayout;
	Discrete_Image.NodeState:=NodeState;
	
	Discrete_Image.Input_Node_Count:= Discrete_In.Input_Node_Count;
	Discrete_Image.VB_Node_Count:= Discrete_In.VB_Node_Count;
	Discrete_Image.Water_Stand_Count:= Discrete_In.Water_Stand_Count;

	IF  (Discrete_Image.Input_Node_Count < 4)
		THEN Discrete_Image.VB_Screen_Position:= 1;
	ELSIF  (Discrete_Image.Input_Node_Count < 7)
		THEN Discrete_Image.VB_Screen_Position:= 2;
	ELSIF  (Discrete_Image.Input_Node_Count < 10)
		THEN Discrete_Image.VB_Screen_Position:= 3;
	ELSIF  (Discrete_Image.Input_Node_Count < 13)
		THEN Discrete_Image.VB_Screen_Position:= 4;
	ELSIF  (Discrete_Image.Input_Node_Count < 16)
		THEN Discrete_Image.VB_Screen_Position:= 5;
	ELSIF  (Discrete_Image.Input_Node_Count < 19)
		THEN Discrete_Image.VB_Screen_Position:= 6;
	ELSIF  (Discrete_Image.Input_Node_Count < 22)
		THEN Discrete_Image.VB_Screen_Position:= 7;
	ELSIF  (Discrete_Image.Input_Node_Count < 26)
		THEN Discrete_Image.VB_Screen_Position:= 8;
	ELSE
			Discrete_Image.VB_Screen_Position:= 9;
	END_IF;

	Discrete_Image.N00:= N00;
	Discrete_Image.N01:= N01;
	Discrete_Image.N02:= N02;
	Discrete_Image.N03:= N03;
	Discrete_Image.N04:= N04;
	Discrete_Image.N05:= N05;
	Discrete_Image.N06:= N06;
	Discrete_Image.N07:= N07;
	Discrete_Image.N08:= N08;
	Discrete_Image.N09:= N09;
	Discrete_Image.N10:= N10;
	Discrete_Image.N11:= N11;
	Discrete_Image.N12:= N12;
	Discrete_Image.N13:= N13;
	Discrete_Image.N14:= N14;
	Discrete_Image.N15:= N15;
	Discrete_Image.N16:= N16;
	Discrete_Image.N17:= N17;
	Discrete_Image.N18:= N18;
	Discrete_Image.N19:= N19;
	Discrete_Image.N100:= N100;
	Discrete_Image.N100_STAT:= N100_STAT;
	Discrete_Image.N101:= N101;
	Discrete_Image.N101_STAT:= N101_STAT;
	Discrete_Image.N102:= N102;
	Discrete_Image.N102_STAT:= N102_STAT;
	
	(*IsEnabled control For UI screen: Default "IsEnabled == True"*)
	Discrete_Image.Enable_FixtureContext_Clamps:= TRUE;
	Discrete_Image.Enable_FixtureContext_QA:= TRUE;
	Discrete_Image.Enable_FixtureContext_Manual:= TRUE;

	Discrete_Image.ECatSlave_Cable_Breaks:= ECatSlave_Cable_Breaks;

	Discrete_Image.Operator_Performance_Pen:= Production_Report.Shift_Report[0].Prod_Performance;
END_ACTION

END_PROGRAM

// ---- POUs/FBs/FB_SmartRay_20260119.TcPOU
(*FB for use SmartRay control/monitoring:
	Original Author(s): Will.K of Sodecia GTAC; 
------------------------------------------------------------------------------------------
REVISION NOTES:
	Version 20260119: This function block manages the PLC ↔ SmartRay ↔ KUKA robot inspection handshake sequence.
	                  This version utilizes three signals from the KUKA FB custom inputs (Heartbeat(1 bit), InspectionCompleted(1 bit), and Global Error(1 bit))
                      to control sequencing and fault handling.(Robot-to-PLC signal mapping is required)
                      Synchronizes 'PartType' and 'PartID' between PLC and SmartRay before inspection
                      Provides a 'Robot_Start_Ready' signal once PLC data is validated.
                      Monitors robot inspection start and inspection completion.
                      Evaluates inspection results (OK / NOK) from SmartRay.
                      Monitors communication health via heartbeat supervision.
                      Reports global fault and communication error status.
                      Controls inspection completion and reset sequencing.
                      The inspection result is considered valid only when: 
                      1. Communication is healthy
                      2. PartType and PartID match
                      3. SmartRay signals ResultValid and robot signals InspectionCompleted *)
FUNCTION_BLOCK FB_SmartRay_20260119
VAR_INPUT
	
	In_Robot_From_SR : udt_SmartRay_Out_To_Robot_IN_20260119;
	Out_Robot_To_SR : udt_Robot_Out_To_SmartRay_IN_20260119;
	
	Discrete_In : udt_SRxx_Input_Image ; // from hmi	
	
	Previous_Job_Complete : BOOL; // previous job complete
	Robot_Inspection_Start : BOOL; // Robot calls the jobs

	PartType : BYTE;
	PartID : ARRAY[0..19] OF BYTE;

	
	All_Reset : BOOL;
END_VAR
VAR_OUTPUT
    Discrete_Image : udt_SRxx_DiscreteImage;
	Profinode_OK :BOOL;
	Robot_Start_Ready : BOOL; // robot is okay to start the job, plc job is done
	
	Error : BOOL; // Global Error 
	Comm_Error : BOOL; // Comm Error
	FB_Error : BOOL; // internal fb seq fault
	
END_VAR

VAR_OUTPUT PERSISTENT 
	PLC_Inspection_Complete : BOOL; // robot inspection complete
	Smart_Ray_OK  : BOOL;
	Smart_Ray_NOK : BOOL;
	
END_VAR
VAR

    (*Max Attempt count*)
    Max_Attempt : INT; // Preventing from endless loop
	Attempt_Flag: BOOL;
	
	(*Bypass R_trig*)
	Bypass_R_trig_ON : R_TRIG;
	Bypass_R_trig_OFF: R_TRIG;
 
	FB_OK : BOOL;
	i_step : INT;
	i_Faulted_step: INT;
	i_partid: INT;
	PartID_Match : BOOL;
	PartID_Not_Match : BOOL;
	
	HeartbeatTimer_Robot: TON;
	CommFaulted_Robot: BOOL;
	
	PartID_Check_Start: BOOL;
	PartID_Check_Delay: TON;
	(*Map with Profinet Slave I/O*)
	In_From_SmartRay AT %I* : udt_SmartRay_Out_To_PLC_IN_20260119;
	Out_To_SmartRay AT %Q* : udt_PLC_Out_To_SmartRay_IN_20260119;
	
	(*Status*)
	Internal_ProfiNet AT %I* : udt_ProfiNet_Status;
	

	
    (*PLC Input from Smart Ray*)
	(*#########################*)
	(*Byte 0*)
	In_PartType : BYTE; 
	(*Byte 2-21*)
	In_PartID : ARRAY[0..19] OF BYTE;
	(*Byte 22*)
	In_QualityOK : BOOL; (*Bit 0*)
	In_QualityNOK : BOOL; (*Bit 1*)
	In_ResultValid : BOOL; (*Bit 2*)
	In_LastTelegramSent : BOOL; (*Bit 7*)
	(*Byte 24-43*)
	In_PartIDVisu1 : ARRAY[0..19] OF BYTE;
	(*Byte 44*)
	In_WorkerResultOK : BOOL; (*Bit 0*)
	In_WorkerResultNOK : BOOL; (*Bit 1*)
	In_ReworkOK : BOOL; (*Bit 2*)
	In_ReworkDone : BOOL; (*Bit 3*)
	In_Visu_NextPage : BOOL; (*Bit 4*)
	In_Visu_NextWeld : BOOL; (*Bit 5*)
	In_Visu_PreviousWeld : BOOL; (*Bit 6*)
	(*Byte 45*)
	In_Visu_WorkerButon :BYTE; 
	(*Byte 48-67*)
	In_PartIDVisu2 : ARRAY[0..19] OF BYTE;
	(*Byte 68*)
	In_WorkerResultOK2 : BOOL; (*Bit 0*)
	In_WorkerResultNOK2 : BOOL; (*Bit 1*)
	In_ReworkOK2 : BOOL; (*Bit 2*)
	In_ReworkDone2 : BOOL; (*Bit 3*)
	In_Visu_NextPage2 : BOOL; (*Bit 4*)
	In_Visu_NextWeld2 : BOOL; (*Bit 5*)
	In_Visu_PreviousWeld2 : BOOL; (*Bit 6*)
	(*Byte 69*)
	In_Vis_WorkerButton2 : BYTE;
	(*Byte 80-179*)
	In_WeldResult : ARRAY[0..99] OF BYTE;
	(*#########################*)
	
	(*PLC Output to Smart Ray*)
	(*#########################*)
	(*Byte 0*)
	Out_PartType : BYTE;	
	(*Byte 2-21*)
	Out_PartID : ARRAY[0..19] OF BYTE;
	(*Byte 24-43*)
	Out_PartIDVisu1 : ARRAY[0..19] OF BYTE;
	(*Byte 44*)
	Out_Visu_NextPage : BOOL; (*Bit 4*)
	Out_Visu_NextWeld : BOOL; (*Bit 5*)
	Out_Visu_PreviousWeld : BOOL; (*Bit 6*)
	(*Byte 45*)
	Out_Visu_WorkerButton : BYTE; 
	(*Byte 48-67*)
	Out_PartIDVisu2 : ARRAY[0..19] OF BYTE;
	(*Byte 68*)
	Out_Visu_NextPage2 : BOOL; (*Bit 4*)
	Out_Visu_NextWeld2 : BOOL; (*Bit 5*)
	Out_Visu_PreviousWeld2 : BOOL; (*Bit 6*)
	(*Byte 69*)
	Out_Visu_WorkerButton2 : BYTE;
	(*#########################*)

END_VAR

FB_OK := TRUE; (*true if fb is called*)

(*Invoke Inputs/Outputs*)
Inputs();
Outputs();

(*Gather Status Of Hardware*)
IF Internal_ProfiNet.PnIoBoxState = 0
	THEN
	Profinode_OK := TRUE;
ELSE Profinode_OK := FALSE;
END_IF

(*Global Error*)
Error := In_Robot_From_SR.FailureGlobal_Out;

(*Comm status*)
HeartbeatTimer_Robot(IN:= NOT In_Robot_From_SR.Alive_Out, PT:= T#2S);
IF HeartbeatTimer_Robot.Q
	THEN
	CommFaulted_Robot := TRUE;
ELSE CommFaulted_Robot := FALSE;
END_IF
(*Comm Error*)
Comm_Error := CommFaulted_Robot;

(*--------*)
IF Previous_Job_Complete AND NOT PLC_Inspection_Complete AND NOT Discrete_In.Bypass
	THEN
	
	CASE i_step OF 
	0: // Part type 
	   Out_PartType := PartType;
	   IF Out_PartType = In_PartType
		   THEN
		   i_step := 1;
	   END_IF
	1: // Part ID
	   Out_PartID := PartID;
	   	 
       PartID_Check_Delay.PT := T#0.5S;
       PartID_Check_Delay();
	   PartID_Check_Delay.IN := TRUE;
	   
	   PartID_Check_Start:= PartID_Check_Delay.Q;
	   
	   IF PartID_Check_Start AND Max_Attempt <5 // you can change the max attempt number
		   THEN
		   FOR i_partid := 0 TO 19 BY 1 DO
		        IF (Out_PartID[i_partid] <> In_PartID[i_partid])
			          THEN
			          PartID_Match := FALSE;
			          PartID_Not_Match := TRUE;
                      Attempt_Flag := TRUE;				 
			          EXIT;
		        ELSE PartID_Match := TRUE;  
                     PartID_Not_Match := FALSE; 
		        END_IF   
	       END_FOR
	   ELSIF Max_Attempt >= 5
		       THEN
			   i_Faulted_step := i_step;
		       i_step := 100; 	   
	   END_IF
	   
	   IF Attempt_Flag
		   THEN
		   Max_Attempt := Max_Attempt + 1;
		   Attempt_Flag := FALSE;
	   END_IF
	   
	   IF PartID_Match AND NOT PartID_Not_Match
		   THEN
		   PartID_Check_Delay.IN := FALSE;
		   IF NOT PartID_Check_Delay.Q
			   THEN
			   i_step := 2;   
		   END_IF

	   END_IF
	   
	2:  // plc signal update is done, robot can start the job
	   Robot_Start_Ready := TRUE;
	   
	   IF Robot_Inspection_Start
		   THEN 
		   i_step :=3; // robot called the jobs 
	   END_IF
	   
	3: // wait for the result 
	   IF In_ResultValid AND Out_Robot_To_SR.InspectionCompleted_In
		   THEN
		   Smart_Ray_OK := In_QualityOK;
		   Smart_Ray_NOK := In_QualityNOK; 
		   i_step :=4;
	   END_IF
	   
	 4: 
	   IF (Smart_Ray_OK = In_QualityOK) AND 
          (Smart_Ray_NOK = In_QualityNOK)
            THEN
			i_step :=5;
       END_IF 
	    
	5: // Complete 
       PLC_Inspection_Complete := TRUE;  
	   
	100: // Internal seq error  
        FB_Error := TRUE;  
		
		IF Discrete_In.Retry // from HMI
            THEN
            FB_Error := FALSE;
            Max_Attempt := 0;
            Attempt_Flag := FALSE;
            PartID_Match := FALSE;
            PartID_Not_Match := FALSE;
            PartID_Check_Delay.IN := FALSE;
            i_step := 0;
        END_IF
   
    END_CASE

END_IF
(*--------*)

(*Bypass*)
Bypass_R_trig_ON.CLK := Discrete_In.Bypass ;
Bypass_R_trig_ON();
IF Bypass_R_trig_ON.Q 
	THEN
	Robot_Start_Ready := TRUE;  
    Smart_Ray_OK := TRUE;      
    Smart_Ray_NOK := FALSE;
    PLC_Inspection_Complete := TRUE;
    i_step := 0;
END_IF

Bypass_R_trig_OFF.CLK := NOT Discrete_In.Bypass ;
Bypass_R_trig_OFF();
IF Bypass_R_trig_OFF.Q 
	THEN
	Robot_Start_Ready := FALSE;  
    Smart_Ray_OK := FALSE;      
    Smart_Ray_NOK := FALSE;
    PLC_Inspection_Complete := FALSE;
END_IF

(*Reset*)
IF PLC_Inspection_Complete AND All_Reset
	THEN
	Robot_Start_Ready := FALSE;
	PLC_Inspection_Complete := FALSE;
	PartID_Check_Start := FALSE;
	Smart_Ray_OK  := FALSE;
	Smart_Ray_NOK  := FALSE;
	PartID_Match := FALSE;
	PartID_Not_Match := FALSE;
	i_step := 0;
	i_Faulted_step := 0;
	Max_Attempt := 0;
	Attempt_Flag := FALSE;

END_IF


(*Discrete image*)
Discrete_Image.Profinode_status:= Internal_ProfiNet;
Discrete_Image.SR_Comm_Error := CommFaulted_Robot;
Discrete_Image.SR_Error := Error;
Discrete_Image.SR_PLC_FB_Error := FB_Error;
Discrete_Image.SR_Smart_Ray_OK := Smart_Ray_OK;
Discrete_Image.SR_Smart_Ray_NOK := Smart_Ray_nOK;

ACTION Inputs:
(*Mapping Information Convertion*)

 (*Smart Ray to PLC*)
	(*Byte 0*)
	In_PartType := In_From_SmartRay.Byte_0; 
	(*Byte 2-21*)
	In_PartID := In_From_SmartRay.Byte_2_21;
	(*Byte 22*)
	In_QualityOK := In_From_SmartRay.Byte_22.0; (*Bit 0*)
	In_QualityNOK := In_From_SmartRay.Byte_22.1; (*Bit 1*)
	In_ResultValid := In_From_SmartRay.Byte_22.2; (*Bit 2*)
	In_LastTelegramSent := In_From_SmartRay.Byte_22.7; (*Bit 7*)
	(*Byte 24-43*)
	In_PartIDVisu1 := In_From_SmartRay.Byte_24_43;
	(*Byte 44*)
	In_WorkerResultOK := In_From_SmartRay.Byte_44.0; (*Bit 0*)
	In_WorkerResultNOK := In_From_SmartRay.Byte_44.1; (*Bit 1*)
	In_ReworkOK := In_From_SmartRay.Byte_44.2; (*Bit 2*)
	In_ReworkDone := In_From_SmartRay.Byte_44.3; (*Bit 3*)
	In_Visu_NextPage := In_From_SmartRay.Byte_44.4; (*Bit 4*)
	In_Visu_NextWeld := In_From_SmartRay.Byte_44.5; (*Bit 5*)
	In_Visu_PreviousWeld := In_From_SmartRay.Byte_44.6; (*Bit 6*)
	(*Byte 45*)
	In_Visu_WorkerButon := In_From_SmartRay.Byte_45; 
	(*Byte 48-67*)
	In_PartIDVisu2 := In_From_SmartRay.Byte_48_67 ;
	(*Byte 68*)
	In_WorkerResultOK2 := In_From_SmartRay.Byte_68.0; (*Bit 0*)
	In_WorkerResultNOK2 := In_From_SmartRay.Byte_68.1; (*Bit 1*)
	In_ReworkOK2 := In_From_SmartRay.Byte_68.2; (*Bit 2*)
	In_ReworkDone2 := In_From_SmartRay.Byte_68.3; (*Bit 3*)
	In_Visu_NextPage2 := In_From_SmartRay.Byte_68.4; (*Bit 4*)
	In_Visu_NextWeld2 := In_From_SmartRay.Byte_68.5; (*Bit 5*)
	In_Visu_PreviousWeld2 := In_From_SmartRay.Byte_68.6; (*Bit 6*)
	(*Byte 69*)
	In_Vis_WorkerButton2 := In_From_SmartRay.Byte_69;
	(*Byte 80-179*)
	In_WeldResult := In_From_SmartRay.Byte_80_179;

(*end*)
END_ACTION

ACTION Outputs:
(*Mapping Information Convertion*)

 (*PLC to Smart Ray*)
    (*Byte 0*)
	Out_To_SmartRay.Byte_0 := Out_PartType;	
	(*Byte 2-21*)
	Out_To_SmartRay.Byte_2_21 := Out_PartID;
	(*Byte 24-43*)
	Out_To_SmartRay.Byte_24_43 := Out_PartIDVisu1;
	(*Byte 44*)
	Out_To_SmartRay.Byte_44.4 := Out_Visu_NextPage; (*Bit 4*)
	Out_To_SmartRay.Byte_44.5 := Out_Visu_NextWeld; (*Bit 5*)
	Out_To_SmartRay.Byte_44.6 := Out_Visu_PreviousWeld; (*Bit 6*)
	(*Byte 45*)
	Out_To_SmartRay.Byte_45 := Out_Visu_WorkerButton; 
	(*Byte 48-67*)
	Out_To_SmartRay.Byte_48_67 := Out_PartIDVisu2;
	(*Byte 68*)
	Out_To_SmartRay.Byte_68.4 := Out_Visu_NextPage2; (*Bit 4*)
	Out_To_SmartRay.Byte_68.5 := Out_Visu_NextWeld2; (*Bit 5*)
	Out_To_SmartRay.Byte_68.6 := Out_Visu_PreviousWeld2; (*Bit 6*)
	(*Byte 69*)
	Out_To_SmartRay.Byte_69 := Out_Visu_WorkerButton2;
	
(*end*)
END_ACTION

END_FUNCTION_BLOCK

// ---- POUs/FBs/FB_GTAC_IV3_20250730.TcPOU
(*FB for use with Keyence IV2 Sensors

------------------------------------------------------------------------------------------
REVISION NOTES:
	Version 20210201: February 1st, 2021
		- Initial Concept (C.Drees)
	
	Version20211109: November 9th, 2021
		- Modified to handle ECAT Layout
	
	Version20211229: December 29th, 2021
		- Added Discrete Node OK Status, j.underhill
		
	Version20220119: January 19th, 2022
		- Added In Auto Status to Control Automated Program Selection, j.underhill
		- Automated Program Selection to IV2 Controller, j.underhill
		
	Version20240315: March 15th, 2024
		- Added "busy" Bit mirror to outputs for program selection backcheck, D Klaassen
		- Added "ProgramSwitchComplete" to outputs for fast switching applications
		- Added Current program to externally track which porgram is running
		
	Version20250725: July 25th, 2025
	    - Automatic retry bit is addded 
*)

FUNCTION_BLOCK FB_GTAC_IV3_20250730
VAR_INPUT
	TriggerRequest: BOOL;			(*Boolean Input to issue a start capture trigger*)
	WarningClear: BOOL;				(*Boolean to clear any warnings on IV2 system*)
	ProgramSwitchRequest: BOOL;		(*Boolean to request a program change *)
	ProgramRequest: INT;			(*Integer between 0 and 31 to switch the program to*)
	BufferClear: BOOL;				(*Boolean to Clear Buffer, used to clear the I/O status from IV2 System*)
	Reset_Sequence: BOOL;			(*Boolean to Reset the Sequence *)
	In_Auto: BOOL;					(*Boolean to check status of Auto Mode*)
	Discrete_In: udt_IVxx_Input_Image_20250812;

END_VAR

VAR_OUTPUT
	IV_Check_OK: BOOL;				(*Camera Check Judgement OK*)
	IV_Check_NOK: BOOL;				(*Camera Check Judgement Not OK *)
	Camera_Faulted: BOOL;			(*Camera Sequence Faulted *)
	Camera_Complete :BOOL;			(*Camera Sequence Complete*)
	Discrete_Image:	udt_IV2_DiscreteImage;
	ProgramSwitchComplete : BOOL; 	(* Camera Check for the program select *)
	Tool_1_out: BOOL; 				(*Tool 1 Out feedback*)
	Tool_2_out: BOOL; 				(*Tool 2 Out feedback*)
	Tool_3_out: BOOL; 				(*Tool 3 Out feedback*)
	Tool_4_out: BOOL; 				(*Tool 4 Out feedback*)
	Tool_5_out: BOOL; 				(*Tool 5 Out feedback*)
	Tool_6_out: BOOL; 				(*Tool 6 Out feedback*)
	Tool_7_out: BOOL; 				(*Tool 7 Out feedback*)
	Tool_8_out: BOOL; 				(*Tool 8 Out feedback*)
	Tool_9_out: BOOL; 				(*Tool 9 Out feedback*)
	Tool_10_out: BOOL; 				(*Tool 10 Out feedback*)
	Tool_11_out: BOOL; 				(*Tool 11 Out feedback*)
	Tool_12_out: BOOL; 				(*Tool 12 Out feedback*)
	Tool_13_out: BOOL; 				(*Tool 13 Out feedback*)
	
	Logic_1_out :BOOL;
	Logic_2_out :BOOL;
	Logic_3_out :BOOL;
	Logic_4_out :BOOL;
	

	
	Result_Available: BOOL;						(*Response from IV2 when a result is ready*)
	CurrentPrg_Out: INT;			(*Shows the Current program running on the unit*)
	IV_Busy_Out: BOOL;
	IV_Running_Outdr:BOOL;
	Faulted: BOOL;
	
	
END_VAR

VAR
	DiscreteNode_OK: BOOL;
	PortB_MissingLink: BOOL;
	ECAT_Input_Data AT %I*: udt_IV2_Inputs;	(*Input image array  EtherCAT*)	
	ECAT_Output_Data AT %Q*:ARRAY[0..5]OF DWORD; 		(*Output Image Array EtherCAT*)

	EIP_Input_Integer AT %I*:ARRAY [0..196] OF INT;		(*Input image array  ETHERNET/IP*)
	EIP_Output_Integer AT %Q*: ARRAY [0..6] OF INT;		(*Output Image Array ETHERNET/IP*)

	TriggerResponse: BOOL;						(*Response from IV2 when triggered*)
	IV_Busy: BOOL;								(*Response from IV2 when processing an image*)
	IV_Running: BOOL;							(*IV2 Running Status *)
	IV_Ready: BOOL;								(*IV2 Ready to Run Status*)
	IV_Warning: BOOL;							(*IV2 Warning, see warning Code*)
	IV_Error: BOOL;								(*IV2 Error, See Error Code*)
	Judgement_OK: BOOL;							(*IV2 Status, all Judgement Code OK *)
	Logic1_OK: BOOL;								(*IV2 Logic 1 Judgement Code OK*)
	Logic2_OK: BOOL;								(*IV2 Logic 2 Judgement Code OK*)
	Logic3_OK: BOOL;								(*IV2 Logic 3 Judgement Code OK*)
	Logic4_OK: BOOL;								(*IV2 Logic 4 Judgement Code OK*)
	TOOL_OK:ARRAY [1..16] OF BOOL;				(*IV2 Boolean status of Pass fail for individual Tools*)
	ProgramSwitch:BOOL;							(*IV2 Program Switch requested*)

	CurrentPrg: INT;								(*IV2 Current Program Running *)
	IV_Sequence: INT;							(*IV2 Sequence Step
													0-  IV2 Not Ready
													10-  IV2 is waiting for a trigger
													20 - Wait for IV2 to be Busy Processing Image
													30 - Wait for  IV2 to be finished processing
													40 - Wait for  IV2 Trigger Response OK and not Failed
													50 - Wait for IV2 to have a Result Available
													60 - Pass/Fail based on Judgement Critera
													70 - Sequence Complete
												*)
	TriggerFail: BOOL;								(*IV2 Trigger Failed Response*)
	ProgramSwitchTON: TON;
	ProgramSwitchTON2: TON;
	FailureRecovery_Attempt : INT; 
    Failure_Max_Attempt_Fault : BOOL ; 
	Fault_Failure_Recovery_Tmrs: ARRAY [1..15] OF TON;
	Fault_Delay: TIME:=T#2.5S;
	Failure_Recovery_Seq : INT; (*Step indication*)
	Fault_Failure_Recovery : ARRAY[1..15] OF BOOL; 
    Failure_Recovery_Trial : BOOL;
	Failure_Recovery_Trigger : BOOL; 
	Failure_R_trig : R_TRIG;
	Failure_Recovery_Delay : TON; (*a bit of delay for re trigger the other cam shots*)
	

END_VAR

(*Discrete I/O Node*)
IF (ECAT_Input_Data.InfoData.State=8)
	THEN DiscreteNode_OK:=TRUE;
ELSE DiscreteNode_OK:=FALSE;
END_IF;

(*Develop Port Connection Warning Flags*)
IF (ECAT_Input_Data.InfoData.State= 9224) (*State Machine for Link Missing at Port B*)
	THEN PortB_MissingLink:= TRUE; (*PortB is OUT Port*)
ELSE PortB_MissingLink := FALSE;
END_IF;

(*I/O Mapping from SM to internal Variables *)
TriggerResponse:= EIP_Input_Integer[0].0 OR ECAT_Input_Data.TriggerResponse ;
Result_Available:=EIP_Input_Integer[1].0 OR ECAT_Input_Data.ResultAvailable;
IV_Busy:=EIP_Input_Integer[1].2 OR ECAT_Input_Data.Busy;
IV_Running:=EIP_Input_Integer[1].3 OR ECAT_Input_Data.Running;
IV_Ready:=EIP_Input_Integer[1].4 OR ECAT_Input_Data.TriggerReady;
TriggerFail:=EIP_Input_Integer[1].8 OR ECAT_Input_Data.TriggerFailed;
IV_Warning:=EIP_Input_Integer[1].14;
IV_Error:=EIP_Input_Integer[1].15 OR ECAT_Input_Data.Error_Status;


Judgement_OK:=EIP_Input_Integer[2].0 OR ECAT_Input_Data.OverallJudgementOK;
Logic1_OK:= Logic_1_out := EIP_Input_Integer[2].2 OR ECAT_Input_Data.LogicResult[1];
Logic2_OK:= Logic_2_out := EIP_Input_Integer[2].3 OR ECAT_Input_Data.LogicResult[2];
Logic3_OK:= Logic_3_out := EIP_Input_Integer[2].4 OR ECAT_Input_Data.LogicResult[3];
Logic4_OK:= Logic_4_out := EIP_Input_Integer[2].5 OR ECAT_Input_Data.LogicResult[4];

Tool_OK[1]:= Tool_1_out := EIP_Input_Integer[3].0 OR ECAT_Input_Data.ToolResult[1];
Tool_OK[2]:= Tool_2_out := EIP_Input_Integer[3].1 OR ECAT_Input_Data.ToolResult[2];
Tool_OK[3]:= Tool_3_out := EIP_Input_Integer[3].2 OR ECAT_Input_Data.ToolResult[3];
Tool_OK[4]:= Tool_4_out := EIP_Input_Integer[3].3 OR ECAT_Input_Data.ToolResult[4];
Tool_OK[5]:= Tool_5_out := EIP_Input_Integer[3].4 OR ECAT_Input_Data.ToolResult[5];
Tool_OK[6]:= Tool_6_out := EIP_Input_Integer[3].5 OR ECAT_Input_Data.ToolResult[6];
Tool_OK[7]:= Tool_7_out :=EIP_Input_Integer[3].6 OR ECAT_Input_Data.ToolResult[7];
Tool_OK[8]:= Tool_8_out :=EIP_Input_Integer[3].7 OR ECAT_Input_Data.ToolResult[8];
Tool_OK[9]:= Tool_9_out :=EIP_Input_Integer[3].8 OR ECAT_Input_Data.ToolResult[9];
Tool_OK[10]:= Tool_10_out :=EIP_Input_Integer[3].9 OR ECAT_Input_Data.ToolResult[10];
Tool_OK[11]:= Tool_11_out :=EIP_Input_Integer[3].10 OR ECAT_Input_Data.ToolResult[11];
Tool_OK[12]:= Tool_12_out :=EIP_Input_Integer[3].11 OR ECAT_Input_Data.ToolResult[12];
Tool_OK[13]:= Tool_13_out :=EIP_Input_Integer[3].12 OR ECAT_Input_Data.ToolResult[13];
Tool_OK[14]:= EIP_Input_Integer[3].13;	(*ECAT Not capable of Data*)
Tool_OK[15]:= EIP_Input_Integer[3].14;	(*ECAT Not capable of Data*)
Tool_OK[16]:= EIP_Input_Integer[3].15;	(*ECAT Not capable of Data*)

IF EIP_Input_Integer[8] > 0 THEN
	CurrentPrg:=EIP_Input_Integer[8];
ELSIF ECAT_Input_Data.ProgramNumber > 0 THEN
	CurrentPrg.0:= ECAT_Input_Data.ProgramNumber.0;
	CurrentPrg.1:= ECAT_Input_Data.ProgramNumber.1;
	CurrentPrg.2:= ECAT_Input_Data.ProgramNumber.2;
	CurrentPrg.3:= ECAT_Input_Data.ProgramNumber.3;
	CurrentPrg.4:= ECAT_Input_Data.ProgramNumber.4;
	CurrentPrg.5:= ECAT_Input_Data.ProgramNumber.5;
	CurrentPrg.6:= ECAT_Input_Data.ProgramNumber.6;
ELSE
	CurrentPrg:=0;
END_IF

(*IO Mapping from Internal Variables to SM*)
EIP_Output_Integer[0].0 := ECAT_Output_Data[1].2:= TriggerRequest;
EIP_Output_Integer[0].2 := ECAT_Output_Data[1].1:= ProgramSwitch;
EIP_Output_Integer[0].3 := ECAT_Output_Data[1].6:= WarningClear;
EIP_Output_Integer[0].5 := ECAT_Output_Data[1].5:= BufferClear;
EIP_Output_Integer[2] := ProgramRequest;

ECAT_Output_Data[2].1:=ProgramRequest.0;
ECAT_Output_Data[3].1:=ProgramRequest.1;
ECAT_Output_Data[4].1:=ProgramRequest.2;
ECAT_Output_Data[5].1:=ProgramRequest.3;



(*Camera Sequence*)
CASE IV_Sequence OF

	0: (*Wait for IV2 Camera to be ready *)

		IF TriggerRequest THEN  (*NOTE: IF the trigger Request is kept on sequence can't start, the sequence must see a Rising edge on the "Trigger Request" *)
			IV_Sequence:=999;
		END_IF

		IF IV_Running  AND NOT TriggerRequest THEN
			IV_Sequence := 10;
		END_IF

	10: (*Wait for Trigger from Main Program Call *)
		IF TriggerRequest THEN
			IV_Sequence :=20;
		END_IF

	20: (*Wait for IV camera to be busy Processing the Image*)
		IF IV_Busy THEN
			IV_Sequence :=30;
			IV_Busy_Out :=IV_Busy;
		END_IF

(*		IF NOT TriggerRequest THEN	(* "Trigger Request" must stay high during entire busy sequence*)
			IV_Sequence:=999;
		END_IF

*)	30:(*Wait for IV Camera to be finished Processing the Image*)
		IF NOT IV_Busy THEN
			IV_Busy_Out := IV_Busy;
			IV_Sequence :=40;
		END_IF

(*		IF NOT TriggerRequest THEN (* "Trigger Request" must stay high during entire busy sequence*)
			IV_Sequence:=999;
		END_IF
*)

	40:(*Verify that the trigger did not fail to take an image*)
		IF  NOT TriggerFail THEN
			IV_Sequence:=50;
		END_IF

		IF TriggerFail THEN  (*If the Trigger failed throw an FB Error *)
			IV_Sequence :=999;
		END_IF

	50:(*Wait for a result to be available*)
		IF Result_Available THEN
			IV_Sequence :=60;
		END_IF

	60:(*Set Pass/Fail based on Overall Judgement status*)
		IF Judgement_OK THEN
			IV_Check_OK := TRUE;
			IV_Check_NOK :=FALSE;
			IV_Sequence:=70;
		ELSE
			IV_Check_NOK := TRUE;
			IV_Check_OK :=FALSE;
			IV_Sequence:=70;
		END_IF

	70:(*Set Camera Sequence Complete*)
		Camera_Complete:=TRUE;


	999: (*If any failure or fault occurs during the sequence, turn on the Camera Faulted bit*)
		Camera_Faulted :=TRUE;
		(*IF Judgement_OK THEN
			IV_Sequence :=60;
		END_IF*)

END_CASE


	(*If a Reset Sequence request turns on, reset the Sequence to 0*)
	IF Reset_Sequence THEN
		IV_Sequence:=0;
		Camera_Complete:= FALSE;
		Camera_Faulted:= FALSE;
	END_IF

	(*Reset Pass/Fail/Complete Bits if the sequence isn't complete*)
	IF IV_Sequence <> 70 THEN
		IV_Check_NOK := FALSE;
		IV_Check_OK :=FALSE;
		Camera_Complete:=FALSE;
	END_IF
	
	(*Reset Fault on IV2 Controller*)
	IF WarningClear THEN
		Camera_Faulted:= FALSE;
	END_IF

	(*If a Program Switch is requested, and is required then issue a program switch to the IV2*)

ProgramSwitchTON(in:=ProgramRequest <> CurrentPrg AND NOT ProgramSwitchTON2.Q,pt:=t#50ms);
ProgramSwitchTON2(in:=ProgramSwitchTON.Q,pt:=T#50MS);

ProgramSwitchRequest:= (ProgramRequest <> CurrentPrg) AND In_Auto;

	IF ProgramSwitchRequest  AND ProgramSwitchTON.q THEN
		IF ProgramRequest <> CurrentPrg  THEN
			ProgramSwitch:=TRUE;
		END_IF
	ELSE
		ProgramSwitch:=FALSE;
	END_IF
	
	IF NOT ProgramSwitch THEN
		ProgramSwitchComplete := TRUE;
	ELSE 
		ProgramSwitchComplete := False;
	END_IF
	CurrentPrg_OUT := CurrentPrg;
	
	(***************************************************************************************)
	(*Auto recovery*)
	IF Discrete_In.FailureRecovery_Enable AND ((FailureRecovery_Attempt) >= (Discrete_In.FailureRecovery_Attempt_Max)) 
       AND IV_Check_NOK 
	   THEN 
	   FailureRecovery_Attempt := FailureRecovery_Attempt + 1;
	   Failure_Recovery_Seq := 1;
	END_IF
	
	Failure_R_trig(CLK:=Failure_Recovery_Trial , Q=> );
	IF Failure_R_trig.Q 
		THEN 
		Reset_Sequence := TRUE;
		Failure_Recovery_Seq :=2;
	END_IF
	
	IF Reset_Sequence AND Failure_Recovery_Trial 
		THEN
		Failure_Recovery_Trigger := TRUE;
		Failure_Recovery_Trial := FALSE;
		Reset_Sequence := FALSE;
		Failure_Recovery_Seq :=3;
		
	END_IF

	Failure_Recovery_Delay(IN:=Failure_Recovery_Trigger , PT:= T#1.5S , Q=> , ET=> ); (*PT time need to be changed based on how many tools are used on cam program to spilt out the result*)	
	IF Failure_Recovery_Delay.Q 
		THEN 
		TriggerRequest := TRUE;
		Failure_Recovery_Trigger := FALSE;	
		Failure_Recovery_Seq :=4;
	END_IF
	
	IF (IV_Check_OK AND Camera_Complete) OR Discrete_In.IVx_Release  
        THEN
		Failure_Recovery_Seq :=0;
		FailureRecovery_Attempt  := 0;
	END_IF	
	
    (*Auto recovery Fault Flags*)
	IF Discrete_In.FailureRecovery_Enable AND (FailureRecovery_Attempt >= Discrete_In.FailureRecovery_Attempt_Max) 
		THEN 
		Failure_Max_Attempt_Fault := TRUE; 
	ELSE 
		Failure_Max_Attempt_Fault := FALSE;
	END_IF
	
	(*auto recovery seq Faults*)
	Fault_Failure_Recovery_Tmrs[1].PT := Fault_Delay;
	Fault_Failure_Recovery_Tmrs[1]();
	Fault_Failure_Recovery_Tmrs[1].IN:= (Failure_Recovery_Seq = 1);
	Fault_Failure_Recovery[1] := Fault_Failure_Recovery_Tmrs[1].Q; 
	
	Fault_Failure_Recovery_Tmrs[2].PT := Fault_Delay;
	Fault_Failure_Recovery_Tmrs[2]();
	Fault_Failure_Recovery_Tmrs[2].IN:= (Failure_Recovery_Seq = 2);
	Fault_Failure_Recovery[2] := Fault_Failure_Recovery_Tmrs[2].Q;
	
	Fault_Failure_Recovery_Tmrs[3].PT := Fault_Delay;
	Fault_Failure_Recovery_Tmrs[3]();
	Fault_Failure_Recovery_Tmrs[3].IN:= (Failure_Recovery_Seq = 3);
	Fault_Failure_Recovery[3] := Fault_Failure_Recovery_Tmrs[3].Q;
	
	Fault_Failure_Recovery_Tmrs[4].PT := Fault_Delay;
	Fault_Failure_Recovery_Tmrs[4]();
	Fault_Failure_Recovery_Tmrs[4].IN:= (Failure_Recovery_Seq = 4);
	Fault_Failure_Recovery[4] := Fault_Failure_Recovery_Tmrs[4].Q;

	IF IV_Error OR (ECAT_Input_Data.ErrorCode <> 0) OR TriggerFail OR Failure_Max_Attempt_Fault OR ECAT_Input_Data.NoFreeSpaceSD
		THEN
		Faulted:= TRUE;
		ELSE
		Faulted:= FALSE;
	END_IF
	
	(***************************************************************************************)
	
	Discrete_Image.IV_Check_OK := IV_Check_OK;
	Discrete_Image.IV_Check_NOK := IV_Check_NOK;
	
	Discrete_Image.Faulted:= Faulted;
	Discrete_Image.PortB_MissingLink:= PortB_MissingLink;
	Discrete_Image.Busy:= IV_Busy;
	Discrete_Image.ErrorStatus:=IV_Error;
	Discrete_Image.ErrorCode:=ECAT_Input_Data.ErrorCode;
	Discrete_Image.InfoData:=Ecat_Input_Data.InfoData;
	Discrete_Image.OverallJudgementOK:=Judgement_OK;
	Discrete_Image.ProgramNumber:=CurrentPrg;
	Discrete_Image.ResultAvailable:=Result_Available;
	Discrete_Image.Running:=IV_Running;
	Discrete_Image.TriggerOutput:=EIP_Output_Integer[0].0;
	Discrete_Image.TriggerFailed:=TriggerFail;
	Discrete_Image.TriggerReady:=IV_Ready;
	Discrete_Image.TriggerResponse:=TriggerResponse;
	
	Discrete_Image.Fault_Failure_Recovery:= Fault_Failure_Recovery; 
	Discrete_Image.Failure_Max_Attempt_Fault := Failure_Max_Attempt_Fault;

END_FUNCTION_BLOCK

// ---- POUs/Fixtures and EOAT/Internal/Fix103.TcPOU
(*Fixture*)

PROGRAM Fix103
	VAR_INPUT
		Enable_Prog: BOOL;
		Enable_Motion: BOOL;
		Discrete_In: udt_FixXX_Input_Image_20180202;
		Dry_Cycle: BOOL;
		Cell_In_Services: BOOL;
		Flash_Rate: BOOL;
		NodeLayout:udt_ECATNodeData_20221507;

	END_VAR

	VAR
(*Hardware Related Data Types*)
			(*Develop "Beckhoff Nodes"*)
			{attribute 'OPC.UA.DA':='1'}
			N00 AT %I*: udt_EP1111;
			{attribute 'OPC.UA.DA':='1'}
			N01 AT %I*: udt_EP1008_002_v2;
			{attribute 'OPC.UA.DA':='1'}
			N02 AT %I*: udt_EP1008_002_v2;
			{attribute 'OPC.UA.DA':='1'}
			N03 AT %I*: udt_EP1008_002_v2;
			{attribute 'OPC.UA.DA':='1'}
			N04 AT %I*: udt_EP1008_002_v2;
			{attribute 'OPC.UA.DA':='1'}
			N05 AT %I*: udt_EP1008_002_v2;
			{attribute 'OPC.UA.DA':='1'}
			N06 AT %I*: udt_EP1008_002_v2;
			{attribute 'OPC.UA.DA':='1'}
			N07 AT %I*: udt_EP1008_002_v2;
			{attribute 'OPC.UA.DA':='1'}
			N08 AT %I*: udt_EP1008_002_v2;
			{attribute 'OPC.UA.DA':='1'}
			N09 AT %I*: udt_EP1008_002_v2;
			{attribute 'OPC.UA.DA':='1'}
			N10 AT %I*: udt_EP1008_002_v2;
			{attribute 'OPC.UA.DA':='1'}
			N11 AT %I*: udt_EP1008_002_v2;
			{attribute 'OPC.UA.DA':='1'}
			N12 AT %I*: udt_EP1008_002_v2;
			{attribute 'OPC.UA.DA':='1'}
			N13 AT %I*: udt_EP1008_002_v2;
			{attribute 'OPC.UA.DA':='1'}
			N14 AT %I*: udt_EP1008_002_v2;
			{attribute 'OPC.UA.DA':='1'}
			N15 AT %I*: udt_EP1008_002_v2;
			{attribute 'OPC.UA.DA':='1'}
			N16 AT %I*: udt_EP1008_002_v2;
			{attribute 'OPC.UA.DA':='1'}
			N17 AT %I*: udt_EP1008_002_v2;
			{attribute 'OPC.UA.DA':='1'}
			N18 AT %I*: udt_EP1008_002_v2;
			{attribute 'OPC.UA.DA':='1'}
			N19 AT %I*: udt_EP1008_002_v2;
			{attribute 'OPC.UA.DA':='1'}
			N20 AT %I*: udt_EP1008_002_v2;
			{attribute 'OPC.UA.DA':='1'}
			N21 AT %I*: udt_EP1008_002_v2;
			{attribute 'OPC.UA.DA':='1'}
			N22 AT %I*: udt_EP1008_002_v2;
			{attribute 'OPC.UA.DA':='1'}
			N100 AT %Q*: udt_SMC_EX260_ValveBank;
			{attribute 'OPC.UA.DA':='1'}
			N100_STAT AT %I*:udt_SMC_EX260_Stat;
			{attribute 'OPC.UA.DA':='1'}
			N101 AT %Q*: udt_SMC_EX260_ValveBank;
			{attribute 'OPC.UA.DA':='1'}
			N101_STAT AT %I*:udt_SMC_EX260_Stat;
			{attribute 'OPC.UA.DA':='1'}
			N102 AT %Q*: udt_SMC_EX260_ValveBank;
			{attribute 'OPC.UA.DA':='1'}
			N102_STAT AT %I*:udt_SMC_EX260_Stat;

(* Nodes States*)
		NodeState: ARRAY[0..63] OF UINT;
		DiscreteNode_OK: BOOL;
(*Cable Break States*)
		ECatSlave_Cable_Breaks: ARRAY[0..1] OF DINT;
(*Standard Internal Variables*)
		(*Generic Sensor Variables*)
		All_Sensors_On: UINT;
		All_Sensors_Off: BOOL;
		All_Sensors_Off1: BOOL;
		All_Sensors_Off2: BOOL;
		(*Generic Position Variables*)
		Tool_At_Home: BOOL;
		Tool_At_Load: UINT;
		Tool_At_Weld: UINT;
		Tool_At_Rotate: UINT;
		Tool_At_Seal: UINT;
		Tool_At_Stud: UINT;
		Tool_At_Unload: UINT ;
		(*Grouping Of Items*)
		All_QAChecks_OK: BOOL;
		QAChecks_Failed: BOOL;
		(*General Internals*)
		In_Auto: BOOL;
		In_Manual: BOOL;

		Auto_Run: BOOL;
		Reset_All_Completes:BOOL;
		Load_Robots_Clear1: BOOL;
		Load_Robots_Clear2: BOOL;
		Load_Robots_Clear: BOOL;
		Load_Robots_WorkingOK1: BOOL;
		Load_Robots_WorkingOK2: BOOL;
		Load_Robots_Complete1: BOOL;
		Load_Robots_Complete2: BOOL;
		Load_Robots_PartInEOAT1: BOOL;
		Load_Robots_PartInEOAT2: BOOL;
		Load_Robots_UnclampEarly1: BOOL;
		Load_Robots_UnclampEarly2: BOOL;
		Seal_Robots_Clear: BOOL;
		Seal_Robots_WorkingOK: BOOL;
		Seal_Robots_UnclampEarly: BOOL;
		Seal_Robots_Complete: BOOL;
		Stud_Robots_Clear: BOOL;
		Stud_Robots_WorkingOK: BOOL;
		Stud_Robots_UnclampEarly: BOOL;
		Stud_Robots_Complete: BOOL;
		Weld_Robots_Clear: BOOL;
		Weld_Robots_WorkingOK: BOOL;
		Weld_Robots_UnclampEarly: BOOL;
		Weld_Robots_Complete: BOOL;
		Mig_Robots_Ready :BOOL;
		TurntableA_Clear: BOOL;
		TurntableB_Clear: BOOL;
		Turntable_Clear:BOOL;
		Turntable_WorkingOK: BOOL;
		TurntableA_Complete: BOOL;
		TurntableB_Complete: BOOL;
		Unload_Robots_Clear1: BOOL;
		Unload_Robots_WorkingOK1: BOOL;
		Unload_Robots_Complete1: BOOL;
		Unload_Robots_EOATEmpty1: BOOL;
		Unload_Robots_Clear2: BOOL;
		Unload_Robots_WorkingOK2: BOOL;
		Unload_Robots_Complete2: BOOL;
		Unload_Robots_EOATEmpty2: BOOL;
		Unload_Robots_Clear: BOOL;
		All_Robots_Clear: BOOL;

		Unload_Robot_Complete: BOOL;

		Start_Load_Robots1: BOOL;
		Start_Load_Robots2: BOOL;
		Start_Weld_Robots: BOOL;
		Start_Unload_Robots1: BOOL;
		Start_Unload_Robots2: BOOL;
		Start_Seal_Robots: BOOL;
		Start_Stud_Robots: BOOL;
		Start_TurntableA: BOOL;
		Start_TurntableB: BOOL;
		Load_Robots_Proceed1: BOOL;
		Load_Robots_Proceed2: BOOL;
		Weld_Robots_Proceed: BOOL;
		Seal_Robots_Proceed: BOOL;
		Stud_Robots_Proceed: BOOL;
		Unload_Robots_Proceed1: BOOL;
		Unload_Robots_Proceed2: BOOL;

		Prod_Inc: R_TRIG;
		Cycle_Time: TON;
		Cycle_Time_Pulse: R_TRIG;
		Load_Time: TON;
		Weld_Time: TON;
		Seal_Time: TON;
		Stud_Time: TON;
		Turn_Time: TON;
		Unload_Time: TON;
		Date_Stamp_TMR: TON;
		Date_StampHome_TMR: TON;
		CLFaulted: UDINT;
		PPFaulted: UDINT;
		Manual_Ind_HomePrompt: BOOL;
		Fixture_Allow_Model_Change: BOOL;

(*Non-Standard Variables*)

		(*FB Instances*)
		Clamp1FB: FB_Cylinder_Status;
		Clamp2FB: FB_Cylinder_Status;
		Clamp3FB: FB_Cylinder_Status;
		Clamp4FB: FB_Cylinder_Status;
		Clamp5FB: FB_Cylinder_Status;
		Clamp6FB: FB_Cylinder_Status;
		Clamp7FB: FB_Cylinder_Status;
		Clamp8FB: FB_Cylinder_Status;
		Clamp9FB: FB_Cylinder_Status;
		Clamp10FB: FB_Cylinder_Status;
		Clamp11FB: FB_Cylinder_Status;
		Clamp12FB: FB_Cylinder_Status;
		Clamp13FB: FB_Cylinder_Status;
		Clamp14FB: FB_Cylinder_Status;
		Clamp15FB: FB_Cylinder_Status;
		Clamp16FB: FB_Cylinder_Status;
		Clamp17FB: FB_Cylinder_Status;
		Clamp18FB: FB_Cylinder_Status;
		Clamp19FB: FB_Cylinder_Status;
		Clamp20FB: FB_Cylinder_Status;
		Clamp21FB: FB_Cylinder_Status;
		Clamp22FB: FB_Cylinder_Status;
		Clamp23FB: FB_Cylinder_Status;
		Clamp24FB: FB_Cylinder_Status;
		Cyl1FB: FB_TripleCylinder_20150625;
		Pin1FB: FB_Cylinder_Status;
		Pin2FB: FB_Cylinder_Status;
		Pin3FB: FB_Cylinder_Status;
		Pin4FB: FB_Cylinder_Status;
		Pin5FB: FB_Cylinder_Status;
		Pin6FB: FB_Cylinder_Status;
		Pin7FB: FB_Cylinder_Status;
		Pin8FB: FB_Cylinder_Status;
		Pin9FB: FB_Cylinder_Status;
		Pin10FB: FB_Cylinder_Status;
		Pin11FB: FB_Cylinder_Status;
		Pin12FB: FB_Cylinder_Status;
		Pin13FB: FB_Cylinder_Status;
		Pin14FB: FB_Cylinder_Status;
		Slide1FB: FB_Cylinder_Status;
		Slide2FB: FB_Cylinder_Status;
		Slide3FB: FB_Cylinder_Status;
		Slide4FB: FB_Cylinder_Status;
		Slide5FB: FB_Cylinder_Status;
		Slide6FB: FB_Cylinder_Status;
		Swing1FB: FB_Cylinder_Status;
		Swing2FB: FB_Cylinder_Status;
		Swing3FB: FB_Cylinder_Status;
		Swing4FB: FB_Cylinder_Status;
		Swing5FB: FB_Cylinder_Status;
		Swing6FB: FB_Cylinder_Status;
		QACheck1FB: FB_Cylinder_Status;
		QACheck2FB: FB_Cylinder_Status;
		CheckQA1FB: FB_GTAC_QAcheck_20150529;
		Part_Present1FB: FB_PP_Sensor;
		Part_Present2FB: FB_PP_Sensor;
		Part_Present3FB: FB_PP_Sensor;
		Part_Present4FB: FB_PP_Sensor;
		Part_Present5FB: FB_PP_Sensor;
		Part_Present6FB: FB_PP_Sensor;
		Part_Present7FB: FB_PP_Sensor;
		Part_Present8FB: FB_PP_Sensor;
		Part_Present9FB: FB_PP_Sensor;
		Part_Present10FB: FB_PP_Sensor;
		Part_Present11FB: FB_PP_Sensor;
		Part_Present12FB: FB_PP_Sensor;
		Part_Present13FB: FB_PP_Sensor;
		Part_Present14FB: FB_PP_Sensor;
		Part_Present15FB: FB_PP_Sensor;
		Part_Present16FB: FB_PP_Sensor;
		Part_Present17FB: FB_PP_Sensor;
		Part_Present18FB: FB_PP_Sensor;
		Part_Present19FB: FB_PP_Sensor;
		Part_Present20FB: FB_PP_Sensor;
		Part_Present21FB: FB_PP_Sensor;
		Part_Present22FB: FB_PP_Sensor;
		Part_Present23FB: FB_PP_Sensor;
		Part_Present24FB: FB_PP_Sensor;
		Part_Present25FB: FB_PP_Sensor;
		Part_Present26FB: FB_PP_Sensor;
		Part_Present27FB: FB_PP_Sensor;
		Part_Present28FB: FB_PP_Sensor;
		Part_Present29FB: FB_PP_Sensor;
		Part_Present30FB: FB_PP_Sensor;
		Part_Present31FB: FB_PP_Sensor;
		Part_Present32FB: FB_PP_Sensor;
		Part_Present33FB: FB_PP_Sensor;
		Part_Present34FB: FB_PP_Sensor;
		Part_Present35FB: FB_PP_Sensor;
		Part_Present36FB: FB_PP_Sensor;
		Part_Present37FB: FB_PP_Sensor;
		Part_Present38FB: FB_PP_Sensor;
		Part_Present39FB: FB_PP_Sensor;
		Part_Present40FB: FB_PP_Sensor;
		Tape_Present1FB: FB_PP_Sensor;

		(*Valve FBs*)
		Valve1FB: FB_GTAC_Valve_20170704;
		Valve2FB: FB_GTAC_Valve_20170704;
		Valve3FB: FB_GTAC_Valve_20170704;
		Valve4FB: FB_GTAC_Valve_20170704;
		Valve5FB: FB_GTAC_Valve_20170704;
		Valve6FB: FB_GTAC_Valve_20170704;
		Valve7FB: FB_GTAC_Valve_20170704;
		Valve8FB: FB_GTAC_Valve_20170704;
		Valve9FB: FB_GTAC_Valve_20170704;
		Valve10FB: FB_GTAC_Valve_20170704;
		Valve11FB: FB_GTAC_Valve_20170704;
		Valve12FB: FB_GTAC_Valve_20170704;
		Valve13FB: FB_GTAC_Valve_20170704;
		Valve14FB: FB_GTAC_Valve_20170704;
		Valve15FB: FB_GTAC_Valve_20170704;
		Valve16FB: FB_GTAC_Valve_20170704;
		Valve17FB: FB_GTAC_Valve_20170704;
		Valve18FB: FB_GTAC_Valve_20170704;
		Valve19FB: FB_GTAC_Valve_20170704;
		Valve20FB: FB_GTAC_Valve_20170704;
		Valve21FB: FB_GTAC_Valve_20170704;
		Valve22FB: FB_GTAC_Valve_20170704;
		Valve23FB: FB_GTAC_Valve_20170704;
		Valve24FB: FB_GTAC_Valve_20170704;
		Valve25FB: FB_GTAC_Valve_20170704;
		Valve26FB: FB_GTAC_Valve_20170704;
		Valve27FB: FB_GTAC_Valve_20170704;
		Valve28FB: FB_GTAC_Valve_20170704;
		Valve29FB: FB_GTAC_Valve_20170704;
		Valve30FB: FB_GTAC_Valve_20170704;
		Valve31FB: FB_GTAC_Valve_20170704;
		Valve32FB: FB_GTAC_Valve_20170704;
		Valve33FB: FB_GTAC_Valve_20170704;
		Valve34FB: FB_GTAC_Valve_20170704;
		Valve35FB: FB_GTAC_Valve_20170704;
		Valve36FB: FB_GTAC_Valve_20170704;
		Valve37FB: FB_GTAC_Valve_20170704;
		Valve38FB: FB_GTAC_Valve_20170704;
		Valve39FB: FB_GTAC_Valve_20170704;
		Valve40FB: FB_GTAC_Valve_20170704;
		Valve41FB: FB_GTAC_Valve_20170704;
		Valve42FB: FB_GTAC_Valve_20170704;
		Valve43FB: FB_GTAC_Valve_20170704;
		Valve44FB: FB_GTAC_Valve_20170704;
		Valve45FB: FB_GTAC_Valve_20170704;
		Valve46FB: FB_GTAC_Valve_20170704;
		Valve47FB: FB_GTAC_Valve_20170704;
		Valve48FB: FB_GTAC_Valve_20170704;

		(*Tool Positions*)
			(*Add User Indivdual Position Variables Here*)
			Clamp1ADVD: BOOL;
			Clamp1RETD: BOOL;
			Clamp2ADVD: BOOL;
			Clamp2RETD: BOOL;
			Clamp3ADVD: BOOL;
			Clamp3RETD: BOOL;
			Clamp4ADVD: BOOL;
			Clamp4RETD: BOOL;
			Clamp5ADVD: BOOL;
			Clamp5RETD: BOOL;
			Clamp6ADVD: BOOL;
			Clamp6RETD: BOOL;
			Clamp7ADVD: BOOL;
			Clamp7RETD: BOOL;
			Clamp8ADVD: BOOL;
			Clamp8RETD: BOOL;
			Clamp9ADVD: BOOL;
			Clamp9RETD: BOOL;
			Clamp10ADVD: BOOL;
			Clamp10RETD: BOOL;
			Clamp11ADVD: BOOL;
			Clamp11RETD: BOOL;
			Clamp12ADVD: BOOL;
			Clamp12RETD: BOOL;
			Clamp13ADVD: BOOL;
			Clamp13RETD: BOOL;
			Clamp14ADVD: BOOL;
			Clamp14RETD: BOOL;
			Clamp15ADVD: BOOL;
			Clamp15RETD: BOOL;
			Clamp16ADVD: BOOL;
			Clamp16RETD: BOOL;
			Clamp17ADVD: BOOL;
			Clamp17RETD: BOOL;
			Clamp18ADVD: BOOL;
			Clamp18RETD: BOOL;
			Clamp19ADVD: BOOL;
			Clamp19RETD: BOOL;
			Clamp20ADVD: BOOL;
			Clamp20RETD: BOOL;
			Clamp21ADVD: BOOL;
			Clamp21RETD: BOOL;
			Clamp22ADVD: BOOL;
			Clamp22RETD: BOOL;
			Clamp23ADVD: BOOL;
			Clamp23RETD: BOOL;
			Clamp24ADVD: BOOL;
			Clamp24RETD: BOOL;
			Cyl1ADVD: BOOL;
			Cyl1MID: BOOL;
			Cyl1RETD: BOOL;
			Pin1ADVD: BOOL;
			Pin1RETD: BOOL;
			Pin2ADVD: BOOL;
			Pin2RETD: BOOL;
			Pin3ADVD: BOOL;
			Pin3RETD: BOOL;
			Pin4ADVD: BOOL;
			Pin4RETD: BOOL;
			Pin5ADVD: BOOL;
			Pin5RETD: BOOL;
			Pin6ADVD: BOOL;
			Pin6RETD: BOOL;
			Pin7ADVD: BOOL;
			Pin7RETD: BOOL;
			Pin8ADVD: BOOL;
			Pin8RETD: BOOL;
			Pin9ADVD: BOOL;
			Pin9RETD: BOOL;
			Pin10ADVD: BOOL;
			Pin10RETD: BOOL;
			Pin11ADVD: BOOL;
			Pin11RETD: BOOL;
			Pin12ADVD: BOOL;
			Pin12RETD: BOOL;
			Pin13ADVD: BOOL;
			Pin13RETD: BOOL;
			Pin14ADVD: BOOL;
			Pin14RETD: BOOL;
			Slide1ADVD: BOOL;
			Slide1RETD: BOOL;
			Slide2ADVD: BOOL;
			Slide2RETD: BOOL;
			Slide3ADVD: BOOL;
			Slide3RETD: BOOL;
			Slide4ADVD: BOOL;
			Slide4RETD: BOOL;
			Slide5ADVD: BOOL;
			Slide5RETD: BOOL;
			Slide6ADVD: BOOL;
			Slide6RETD: BOOL;
			Swing1ADVD: BOOL;
			Swing1RETD: BOOL;
			Swing2ADVD: BOOL;
			Swing2RETD: BOOL;
			Swing3ADVD: BOOL;
			Swing3RETD: BOOL;
			Swing4ADVD: BOOL;
			Swing4RETD: BOOL;
			Swing5ADVD: BOOL;
			Swing5RETD: BOOL;
			Swing6ADVD: BOOL;
			Swing6RETD: BOOL;
			QACheck1ADVD: BOOL;
			QACheck1RETD: BOOL;
			QACheck2ADVD: BOOL;
			QACheck2RETD: BOOL;

		(*Part Present Sensors*)
			(*Main Body Present*)
			Part_Present1: BOOL;
			Part_Present2: BOOL;
			Part_Present3: BOOL;
			Part_Present4: BOOL;
			Part_Present5: BOOL;
			Part_Present6: BOOL;
			Part_Present7: BOOL;
			Part_Present8: BOOL;
			Part_Present9: BOOL;
			Part_Present10: BOOL;
			Part_Present11: BOOL;
			Part_Present12: BOOL;
			Part_Present13: BOOL;
			Part_Present14: BOOL;
			Part_Present15: BOOL;
			Part_Present16: BOOL;
			Part_Present17: BOOL;
			Part_Present18: BOOL;
			Part_Present19: BOOL;
			Part_Present20: BOOL;
			Part_Present21: BOOL;
			Part_Present22: BOOL;
			Part_Present23: BOOL;
			Part_Present24: BOOL;
			Part_Present25: BOOL;
			Part_Present26: BOOL;
			Part_Present27: BOOL;
			Part_Present28: BOOL;
			Part_Present29: BOOL;
			Part_Present30: BOOL;
			Part_Present31: BOOL;
			Part_Present32: BOOL;
			Part_Present33: BOOL;
			Part_Present34: BOOL;
			Part_Present35: BOOL;
			Part_Present36: BOOL;
			Part_Present37: BOOL;
			Part_Present38: BOOL;
			Part_Present39: BOOL;
			Part_Present40: BOOL;
			Tape_Present1: BOOL;
			Part_InEOAT04_1_ReadyforThisFix: BOOL; 
			Part_InEOAT04_2_ReadyforThisFix: BOOL; 

		(*Motion Sequence Variables*)
			Clamp_Step: UINT;
			Repo1_Step: UINT;
			Repo2_Step: UINT;
			Repo3_Step: UINT;
			Repo4_Step: UINT;
			Unclamp_Step: UINT;

		(*Custom Application Variables*)
			Weld_Curtain_Bypass: BOOL;
			Vacuum_Bypass: BOOL;
			Sealer_Bypass: BOOL;
			Stud_Bypass: BOOL;
			
			(*Conveyor control*)
			First_Flag: BOOL; (*Finds the first Wall for the index Position*)
			Automatic_Index_CV_Trigger_SR: SR; (*Set for automatic conveyor control*)
			Flag_Watchdog:BOOL; (*Trigger lockout for second flag read*)
			Automatic_Index_CV_Start:BOOL; (*Index Start Command when a part has been loaded *)
			Manual_Index_CV_Trigger_SR : SR; (*Set for HMI trigger*)
			Manual_Index_CV_Start:BOOL; (*Index Start Command when a part has been loaded *)
			Automatic_Stop_Timer : TON; (*Stop signal when a part has been loaded for a few seconds*)
			Manual_Stop_Timer : TON; (*Stop signal if the part has been loaded (detected by the final sensor)*)
			Automatic_Index_CV_Stop : BOOL; (*Stop command that reads the timer*)
			Manual_Index_CV_Stop : BOOL; (*Stop command that reads the timer*)
			Operation_Clear: BOOL; (*Operator Confimation for Indexing Clear*)

			CV_In_Manual : BOOL; (*Conveyor in Manual Operation *)
			CV_In_Auto:BOOL; (*Conveyor in Automatic Operation *)
			CV_Faulted: BOOL; (*Conveyor Faulted *)
			
			HMI_QA_DataGrid: FB_Nok_Datagrid;
		

			(*Force Unload Part button : TCHMI > PLC*)
			Force_Unload_Complete_From_ICxx : ARRAY [0..5] OF BOOL;
            Manual_PartReset_From_ICxx : INT;
			User_Error_Ack_From_ICxx: BOOL;		
		    Current_Nok_Data_Reset_From_ICxx : BOOL;
			History_Nok_Data_Reset_From_ICxx : BOOL;
			Current_History_Reset_From_ICxx : BOOL;
			
			(*PLC > Tchmi*)
			Force_Unload_Part_In_Process_To_ICxx : BOOL; (*Prevents overload reset attempt*)
			Current_Nok_Data_Error_To_ICxx : BOOL;
			History_Nok_Data_Error_To_ICxx : BOOL;
			Force_Unload_Part_Error_To_ICxx : BOOL;
			
			
		
			
			
	Conveyor_Full: BOOL;
END_VAR

	(*data that needs to be retained in the event of a power cycle*)
	VAR PERSISTENT

	
		Load_Complete1: BOOL;
		Load_Complete2: BOOL;
		Load_Complete: BOOL;
		Stud_Complete: BOOL;
		Welding_Complete: BOOL;
		Sealing_Complete: BOOL;
		Unload_Part_Ready : BOOL;
		Unload_Complete: BOOL;
		TurnA_Complete: BOOL;
		TurnB_Complete: BOOL;
		Cycle_Complete: BOOL;
		Eject_Complete: BOOL;
		VacCheck_Complete: BOOL;
		Date_Stamp_Complete: BOOL;
		Load_Seq01: FB_GTAC_Load_Seq_20230302;
		Production_Count:INT;
		Repo_REQS: UINT;
		(*Allow_Load_PreCall: BOOL;
		Allow_Weld_PreCall: BOOL;
		Allow_Unload_PreCall: BOOL;*)
		(*All_SubPP_Off: BOOL;*)
		Production_Report: FB_Production_Report_20221007;
		
		
		Current_Time: DT;
		Current_Time_Str : STRING;
		Current_Time_Len : INT;
	
		(*QA data*)
		Part_Failed_Record : STRING;
        Current_Nok_Data : ARRAY [0..5] OF udt_Generic_Nok_Data_Grid_20251208;
		History_Nok_Data : ARRAY [0..5] OF udt_Generic_Nok_Data_Grid_20251208;
		

	END_VAR

	VAR_OUTPUT

		Prog_Ok: BOOL;
		Discrete_Image: udt_FixXX_Output_Image_20220715;
		In_Auto_Mode: BOOL;
		In_Manual_Mode: BOOL;
		Manual_Indicators1: DINT;
		Manual_Indicators2: DINT;
		Manual_Indicators3: DINT;
		At_Home: BOOL;
		Ready_To_Load: BOOL;
		Red_Lamp_Req: BOOL;
		Status: UINT;
		CLFaults1:UDINT;
		CLFaults2:UDINT;
		CLFaults3:UDINT;
		CLFaults4:UDINT;
		PPFaults: UDINT;
		PPFaults1: UDINT;
		PPFaults2: UDINT;
		Prod_Count_Out: INT;
		Cycle_Time_Out: TIME;
		PrevCycle_Time_Out: TIME;
		Load_Time_Out: TIME;
		Weld_Time_Out: TIME;
		Seal_Time_Out: TIME;
		Stud_Time_Out: TIME;
		Turn_Time_Out: TIME;
		Unload_Time_Out: TIME;
		Model_ID: UINT;
		TurntableA_At_Robot: BOOL;
		TurntableB_At_Robot: BOOL;
		Tool_Call_ForLoadRobots1: BOOL;
		Tool_Call_ForLoadRobots2: BOOL;
		Tool_Call_ForSealRobots: BOOL;
		Tool_Call_ForStudRobots: BOOL;
		Tool_Call_ForWeldRobots: BOOL;
		Tool_Call_ForSweepA: BOOL;
		Tool_Call_ForSweepB: BOOL;
		Tool_Call_ForUnloadRobots1: BOOL;
		Tool_Call_ForUnloadRobots2: BOOL;
		Robots_Clear_ToProceed: BOOL;
		Task_ID: UINT;
		Fix_ID: UINT;
		Load_Complete1_Ack: BOOL;
		Load_Complete2_Ack: BOOL;
		Seal_Complete_Ack: BOOL;
		Stud_Complete_Ack: BOOL;
		Weld_Complete_Ack: BOOL;
		TurnA_Complete_Ack: BOOL;
		TurnB_Complete_Ack: BOOL;
		Unload_Complete1_Ack: BOOL;
		Unload_Complete2_Ack: BOOL;
		Repo_Ack: UINT;
	END_VAR

	(*Set FB_OK to True*)
	Prog_OK:= TRUE;

	(*Conveyor*)
	Conveyor();
	
	
	(*Set conditions to allow model change*)
	Fixture_Allow_Model_Change:= (In_Manual AND Tool_At_Home AND All_Sensors_Off AND All_Robots_Clear)
							OR (Model_ID=0);


	(*Set conditions for interlock Part direction once in EOAT04*)
	(*Welded by all upstream and Failed by Fix102*)
	(*Side 1 of EOAT*)
	Part_InEOAT04_1_ReadyForThisFix:= (EOAT04_1_ProductData_Pers.Generic_PassFail_Notes[1] = 'Comp' 		//Fix01 Weld Comp
									OR EOAT04_1_ProductData_Pers.Generic_PassFail_Notes[2] = 'Comp')		//Fix02 Weld Comp
									AND EOAT04_1_ProductData_Pers.Generic_PassFail_Notes[11] = 'Comp'		//Fix101 Weld Comp
									AND (EOAT04_1_ProductData_Pers.Generic_PassFail_Notes[3] = 'Comp'		//Fix03 Weld Comp
									OR EOAT04_1_ProductData_Pers.Generic_PassFail_Notes[4] = 'Comp')		//Fix04 Weld Comp
									AND (EOAT04_1_ProductData_Pers.Generic_PassFail_Notes[12] = '1' 
											OR EOAT04_1_ProductData_Pers.Generic_PassFail_Notes[12] = '2' 
											OR EOAT04_1_ProductData_Pers.Generic_PassFail_Notes[12] = '3'
											OR EOAT04_1_ProductData_Pers.Generic_PassFail_Notes[12] = 'Fail');  
	//Fix102 Failed : IV3 failed = 1, Smart Ray failed = 2, IV3 & Smart Ray failed = 3
	
	(*Side 2 of EOAT*)
	Part_InEOAT04_2_ReadyForThisFix:= (EOAT04_2_ProductData_Pers.Generic_PassFail_Notes[1] = 'Comp' 		//Fix01 Weld Comp
									OR EOAT04_2_ProductData_Pers.Generic_PassFail_Notes[2] = 'Comp')		//Fix02 Weld Comp
									AND EOAT04_2_ProductData_Pers.Generic_PassFail_Notes[11] = 'Comp'		//Fix101 Weld Comp
									AND (EOAT04_2_ProductData_Pers.Generic_PassFail_Notes[3] = 'Comp'		//Fix03 Weld Comp
									OR EOAT04_2_ProductData_Pers.Generic_PassFail_Notes[4] = 'Comp')		//Fix04 Weld Comp
									AND (EOAT04_2_ProductData_Pers.Generic_PassFail_Notes[12] = '1'
											OR EOAT04_2_ProductData_Pers.Generic_PassFail_Notes[12] = '2' 
											OR EOAT04_2_ProductData_Pers.Generic_PassFail_Notes[12] = '3'
											OR EOAT04_2_ProductData_Pers.Generic_PassFail_Notes[12] = 'Fail');  
	//Fix102 Failed : IV3 failed = 1, Smart Ray failed = 2, IV3 & Smart Ray failed = 3

	(*QA_Data*)
     IF   EOAT04_1_ProductData_Pers.Generic_PassFail_Notes[18] = '1' OR EOAT04_2_ProductData_Pers.Generic_PassFail_Notes[18] = '1'
          THEN
		  Part_Failed_Record := 'IV3 Failed';
	ELSIF EOAT04_1_ProductData_Pers.Generic_PassFail_Notes[18] = '2' OR EOAT04_2_ProductData_Pers.Generic_PassFail_Notes[18] = '2' 	
		  THEN
		  Part_Failed_Record := 'Smart Ray Failed';
	ELSIF EOAT04_1_ProductData_Pers.Generic_PassFail_Notes[18] = '3' OR EOAT04_2_ProductData_Pers.Generic_PassFail_Notes[18] = '3' 	
		  THEN
		  Part_Failed_Record := 'IV3 & Smart Ray Failed';	  
     //ELSE   
    END_IF						
		
  			
(*$$$$$$$$$$$$$$$$$$$$$$$$$$$$$$$$$$$$$$$$$$$$ Fixture Bypasses $$$$$$$$$$$$$$$$$$$$$$$$$$$$$$$$$$$$$$$$$$$$$$$$$$$$*)
	Weld_Curtain_Bypass:= Discrete_In.Bypass_REQS.0;
	Vacuum_Bypass:= Discrete_In.Bypass_REQS.1;
	Stud_Bypass:= Discrete_In.Bypass_REQS.2;
	Sealer_Bypass:= MAIN.SL01.Disp1_Bypass;


(*$$$$$$$$$$$$$$$$$$$$$$$$$$$$$$$$$$$$$$$$$$$$ Gather Status Of Hardware $$$$$$$$$$$$$$$$$$$$$$$$$$$$$$$$$$$$$$$$$$$$$$$$$$$$*)
	(*Check on Status of Hardware*)
	Hardware();

(*$$$$$$$$$$$$$$$$$$$$$$$$$$$$$$$$$$$$$$$$$$$$$ Gather Standard Inputs $$$$$$$$$$$$$$$$$$$$$$$$$$$$$$$$$$$$$$$$$$$$$$$$$$$$$$$$$*)

(*Clamp/Cylinder Inputs*)
	Cylinders();

(*Part Present Inputs*)
	Proxies();


(*$$$$$$$$$$$$$$$$$$$$$$$$$$$$$$$$$$$$$$$$$$$$$$$$ Internal Code $$$$$$$$$$$$$$$$$$$$$$$$$$$$$$$$$$$$$$$$$$$$$$$$$$$$$$$$$$$$$$$$$$$$*)
(*Auto / Manual Mode Code*)
	IF Discrete_In.Mode_Select.0 AND NOT Discrete_In.Mode_Select.1
		THEN
			In_Auto:= TRUE;
			In_Auto_Mode:= TRUE;
	END_IF;
	IF NOT Discrete_In.Mode_Select.0 AND Discrete_In.Mode_Select.1
		THEN
			In_Auto:= FALSE;
			In_Auto_Mode:= FALSE;
	END_IF;
	In_Manual:= NOT In_Auto;
	In_Manual_Mode:= In_Manual;

(*--------------------------------------------------------------------------------Tool Positions---------------------------------------------------------------*)
	Tool_States();

(*----------------------------------------------------Part Present Sensor Input Patterns----------------------------------------------------------------*)
	All_Sensors();


(*>>>>>>>>>>>>>>>>>>>>>>>>>>>>>>>>>>>>>>>>>> Auto Run Cycle >>>>>>>>>>>>>>>>>>>>>>>>>>>>>>>>>>>>>>>*)
(*+++++++++++THIS AREA IS CUSTOM PER INSTALLATION AND WILL HAVE TO BE MODIFIED PER +++++++++++++*)
(*+++++++++++THIS AREA IS CUSTOM PER INSTALLATION AND WILL HAVE TO BE MODIFIED PER +++++++++++++*)
	(*Control of Auto_Run*)
	Auto_Run:= Enable_Motion AND In_Auto AND Model_ID<>0 AND NOT Cycle_Complete;

	(*Auto Run Enables All Other Auto Cycle Code*)
	IF Auto_Run
		THEN

			IF  NOT Load_Complete AND NOT Load_Complete1 AND NOT Automatic_Index_CV_Trigger_SR.Q1 AND NOT Manual_Index_CV_Trigger_SR.Q1
                AND (Part_InEOAT04_1_ReadyForThisFix OR Part_InEOAT04_2_ReadyForThisFix)
				THEN
					(*Start 1st Load Robots*)
					Start_Load_Robots1:= (All_Sensors_Off1 AND (Load_Robots_PartInEOAT1 OR Load_Robots_PartInEOAT2) AND NOT Repo_Reqs.0)
									OR (Repo_Reqs.0 AND All_Sensors_On.0)
									OR Load_Robots_WorkingOK1;
					(*Allow 1st Load Robots To Proceed*)
					Load_Robots_Proceed1:= All_Sensors_Off1 AND (Load_Robots_PartInEOAT1 OR Load_Robots_PartInEOAT2);
			ELSE
					Start_Load_Robots1:= FALSE;
					Load_Robots_Proceed1:= FALSE;
			END_IF;
	

	ELSE
		Start_Load_Robots1:= FALSE;
		Load_Robots_Proceed1:=FALSE;
	END_IF;




(*---------------------------------------------------------------Completes----------------------------------------------------*)
	(*1st Load Complete*)
	IF NOT Dry_Cycle
		THEN
		Load_Complete1:=  All_Sensors_On.0;
	ELSIF Dry_Cycle AND FALSE
		THEN
		IF Tool_At_Home AND Enable_Motion AND All_Sensors_Off
			THEN
			Load_Complete1:= TRUE;
		END_IF;
	END_IF;

	(*All Load Complete*)
	IF NOT Dry_Cycle
		THEN
		Load_Complete:= Load_Complete1 AND Load_Robots_Complete1;
	ELSIF Dry_Cycle AND FALSE
		THEN
		IF Load_Complete1 AND Load_Complete2 AND All_Sensors_Off
			THEN
			Load_Complete:= TRUE;
		END_IF;
	END_IF;
	
	(*Unload Complete*)
	Unload_Part_Ready := (Part_Present5 AND Part_Present6);
	IF (Unload_Part_Ready AND NOT Part_Present5 AND NOT Part_Present6 )
		THEN
		Unload_Complete := TRUE;
		Unload_Part_Ready := FALSE;
	END_IF
	// need feed back to reset the unload complete on conveyor from icxx 
(*!!!!!!!!!!!!!!!!!!!!!!!!!!!!!!!!!!!!!!!!!!!!!!!!!!!!!!!!!!!!!!!!!!!!!!!!!!!!!!!!!!!!!!!!!!!!!!!!! Cycle Complete !!!!!!!!!!!!!!!!!!!!!!!!!!!!!!!!!!!!!!!!!!!!!!!!!!!!!!!!!!!!!!!!!!!!!!!!!!!!!!!!!!!!!!!!!!*)
	(*Set Cycle Complete*)
	IF Auto_Run AND Load_Complete AND All_Robots_Clear
		THEN Cycle_Complete:= TRUE;
	END_IF;
	(*Reset All Completes*)
	IF Load_Robots_Clear
		THEN
			IF In_Manual AND Manual_Index_CV_Start (*this need to be linked into the var of tchmi*) AND All_Sensors_Off1 (*Manual reset => Manual conveyor *)
				THEN
					Reset_All_Completes:= TRUE;
			ELSIF NOT Dry_Cycle AND Cycle_Complete AND All_Sensors_Off1 AND NOT Automatic_Index_CV_Start
				THEN
					Reset_All_Completes:= TRUE;
			ELSIF Dry_Cycle AND Cycle_Complete AND Tool_At_Home AND All_Sensors_Off AND FALSE
				THEN
					Reset_All_Completes:=TRUE;
			ELSE
					Reset_All_Completes:= FALSE;
			END_IF;
	END_IF;
	(*Perform Actual Reset*)
		IF Reset_All_Completes
			THEN
				Cycle_Complete:= FALSE;
				Load_Complete1:= FALSE;
				Load_Complete:= FALSE;
				Load_Robots_UnclampEarly1:= FALSE;
				Load_Robots_UnclampEarly2:= FALSE;
				Repo_Reqs:= 0;
				Reset_All_Completes:= FALSE;
				Part_Failed_Record := '';

		END_IF;

(*---------------------------------------------------------------------------- Call Various Actions ----------------------------------------------------------------------------------------------------*)
	(*Poduction Counters and Report*)
	Production();

	(*Register Robot(s) to Fixture*)
	Robot_Registration();

	(*Setup Fix ID and Model Data*)
	Task_Fix_Model_IDs();

	(*Generate Status Banner and Fault Flags*)
	Status_and_Faults();

	(*Tool Clamp / Unclamp Sequencing and Reposition Handling*)
	Tool_VBSeq_Repos();

	(*Transfer Object Image Data to UI Section*)
	Xfer_To_UI();


(*-----------------------------------------------------------------------------------------Transfer Valve Outputs --------------------------------------------------------------------------------*)
	(*Move "Manual_Home_Prompt" as required for home prompting*)
		Manual_Ind_HomePrompt:= Flash_Rate AND In_Manual AND Discrete_In.Go_Home AND NOT Tool_At_Home;

	(*Call each valve bank*)
	ValveBank1();
	(*ValveBank2();
	ValveBank3(); *)

ACTION All_Sensors:


(*+++++++++++THIS AREA IS CUSTOM PER INSTALLATION AND WILL HAVE TO BE MODIFIED PER +++++++++++++*)
(*+++++++++++THIS AREA IS CUSTOM PER INSTALLATION AND WILL HAVE TO BE MODIFIED PER +++++++++++++*)
(*+++++++++++THIS AREA IS CUSTOM PER INSTALLATION AND WILL HAVE TO BE MODIFIED PER +++++++++++++*)



(**************************************************************************All Sensors Off******************************************************************************)
(**************************************************************************All Sensors Off******************************************************************************)
(**************************************************************************All Sensors Off******************************************************************************)

	(*All Sensors Required Off*)
	All_Sensors_Off:= NOT Part_Present1 AND NOT Part_Present2 AND NOT  Part_Present3
			AND NOT Part_Present4 AND NOT Part_Present5 AND NOT Part_Present6;

	(*All Sensors Required Off - Used for sub fixtures where the part has to move from one stage to the next*)
	All_Sensors_Off1:= NOT Part_Present1 AND NOT Part_Present2;

	(*All Sensors Required Off - Used for sub fixtures where the part has to move from one stage to the next*)
	All_Sensors_Off2:= NOT Part_Present3 AND NOT Part_Present4;



(**************************************************************************All Sensors On******************************************************************************)
(**************************************************************************All Sensors On******************************************************************************)
(**************************************************************************All Sensors On******************************************************************************)


	(*Sensors Required for Start Of 1st Robot Load*)
	All_Sensors_On.0:= Part_Present1 AND Part_Present2;
	(*Sensors Required for Start of 2nd Robot Load*)
	All_Sensors_On.1:= Part_Present3 AND Part_Present4;

	(*Sensors After Load Complete*)
	All_Sensors_On.2:=( Part_Present1 AND Part_Present2 AND Part_Present3
					AND Part_Present4 AND Part_Present5 AND Part_Present6);


	(*Sensors Require for Start Of Welding*)
	All_Sensors_On.3:=(
					((Model_ID=1)
						AND Part_Present1 AND Part_Present2 AND Part_Present3
						AND Part_Present4 AND Part_Present5 AND Part_Present6)

					OR ((Model_ID=2)
						AND Part_Present1 AND Part_Present2 AND Part_Present3
						AND Part_Present4 AND Part_Present5 AND Part_Present6)

					OR ((Model_ID=3)
						AND Part_Present1 AND Part_Present2 AND Part_Present3
						AND Part_Present4 AND Part_Present5 AND Part_Present6)

					OR ((Model_ID=4)
						AND Part_Present1 AND Part_Present2 AND Part_Present3
						AND Part_Present4 AND Part_Present5 AND Part_Present6)
					) OR (All_Sensors_Off AND Dry_Cycle);


	(*Sensors Required After Repo_Reqs.0*)
	All_Sensors_On.4:= (FALSE) OR (Dry_Cycle AND All_Sensors_Off);
	(*Sensors Required After Repo_Reqs.1*)
	All_Sensors_On.5:= (FALSE) OR (Dry_Cycle AND All_Sensors_Off);
	(*Sensors Required After Repo_Reqs.2*)
	All_Sensors_On.6:= (FALSE) OR (Dry_Cycle AND All_Sensors_Off);
	(*Sensors Required After Repo_Reqs.3*)
	All_Sensors_On.7:= (FALSE) OR (Dry_Cycle AND All_Sensors_Off);


	(*Sensors Required for Start Of Unload1*)
	All_Sensors_On.8:=(
					((Model_ID=1)
						AND Part_Present1 AND Part_Present2 AND Part_Present3
						AND Part_Present4 AND Part_Present5 AND Part_Present6)

					OR ((Model_ID=2)
						AND Part_Present1 AND Part_Present2 AND Part_Present3
						AND Part_Present4 AND Part_Present5 AND Part_Present6)

					OR ((Model_ID=3)
						AND Part_Present1 AND Part_Present2 AND Part_Present3
						AND Part_Present4 AND Part_Present5 AND Part_Present6)

					OR ((Model_ID=4)
						AND Part_Present1 AND Part_Present2 AND Part_Present3
						AND Part_Present4 AND Part_Present5 AND Part_Present6)
					) OR (All_Sensors_Off AND Dry_Cycle);

	(*Sensors Required for Start Of Unload2*)
	All_Sensors_On.9:=(
					((Model_ID=1)
						AND Part_Present1 AND Part_Present2 AND Part_Present3
						AND Part_Present4 AND Part_Present5 AND Part_Present6)

					OR ((Model_ID=2)
						AND Part_Present1 AND Part_Present2 AND Part_Present3
						AND Part_Present4 AND Part_Present5 AND Part_Present6)

					OR ((Model_ID=3)
						AND Part_Present1 AND Part_Present2 AND Part_Present3
						AND Part_Present4 AND Part_Present5 AND Part_Present6)

					OR ((Model_ID=4)
						AND Part_Present1 AND Part_Present2 AND Part_Present3
						AND Part_Present4 AND Part_Present5 AND Part_Present6)
					) OR (All_Sensors_Off AND Dry_Cycle);


























(*end*)
END_ACTION

ACTION Conveyor:

	(*Auto / Manual mode*)		
IF In_Auto AND In_Auto_Mode AND NOT CV_In_Manual
    THEN
    CV_In_Auto   := TRUE;
ELSE 
	CV_In_Auto   := FALSE;
END_IF
IF In_Manual AND In_Manual_Mode AND NOT CV_In_Auto
	THEN
	CV_In_Manual := TRUE;
ELSE
	CV_In_Manual := FALSE;
END_IF	

(*Flags and Watchdog*)
First_Flag      := Part_Present1 AND Part_Present2 AND Load_Robots_Complete1;
Flag_Watchdog   := Part_Present3 AND Part_Present4 AND NOT Part_Present1 AND NOT Part_Present2;
Automatic_Index_CV_Trigger_SR.SET1 := First_Flag; 
Automatic_Index_CV_Trigger_SR.RESET := Flag_Watchdog;
Automatic_Index_CV_Trigger_SR();
Operation_Clear := NOT (Part_Present5 AND Part_Present6);

(*Auto Start*) 
IF CV_In_Auto AND Load_Robots_Clear AND Automatic_Index_CV_Trigger_SR.Q1 AND NOT Automatic_Index_CV_Stop
	THEN
	Automatic_Index_CV_Start := TRUE;
ELSE
	Automatic_Index_CV_Start := FALSE;
END_IF
(*Auto Stop*)
Automatic_Stop_Timer.IN := Flag_Watchdog OR NOT Operation_Clear;
Automatic_Stop_Timer.PT := T#4S;
Automatic_Stop_Timer();
IF Automatic_Stop_Timer.Q 
	THEN
	Automatic_Index_CV_Stop := TRUE;
ELSE
	Automatic_Index_CV_Stop := FALSE;
END_IF

(*Manual Control*)
Manual_Index_CV_Trigger_SR.SET1  := Discrete_In.Manual_Conveyor_Start;
Manual_Index_CV_Trigger_SR.RESET := Manual_Index_CV_Stop OR Discrete_In.Go_Home;
Manual_Index_CV_Trigger_SR();

(*Manual Start*)
IF CV_In_Manual AND Load_Robots_Clear AND Manual_Index_CV_Trigger_SR.Q1 AND NOT Manual_Index_CV_Stop
	THEN
	Manual_Index_CV_Start := TRUE; (*stays high untill the part is located on the last sets of proxies*)
ELSE 
	Manual_Index_CV_Start := FALSE;
END_IF
(*Manual Stop*) 
// Manual stop is used when the operator manually drives the part to the last conveyor sensors
Manual_Stop_Timer.IN := NOT Operation_Clear;
Manual_Stop_Timer.PT := T#2S;
Manual_Stop_Timer();
IF Manual_Stop_Timer.Q
	THEN
    Manual_Index_CV_Stop := TRUE;
ELSE
	Manual_Index_CV_Stop := FALSE;
END_IF


Conveyor_Full:= (Part_Present1 AND Part_Present2 AND Part_Present3 AND Part_Present4 AND Part_Present5 AND Part_Present6);

